C01818=1241.105,-36.655,-38.316,-179.706,5.196,148.807
C01819=1241.110,-36.904,-38.303,-179.709,5.195,148.808
C01820=1241.115,-37.154,-38.290,-179.711,5.195,148.809
C01821=1241.121,-37.404,-38.277,-179.714,5.195,148.810
C01822=1241.125,-37.653,-38.263,-179.716,5.196,148.810
C01823=1241.131,-37.903,-38.250,-179.719,5.195,148.811
C01824=1241.135,-38.153,-38.237,-179.721,5.195,148.812
C01825=1241.140,-38.402,-38.224,-179.724,5.195,148.813
C01826=1241.146,-38.651,-38.211,-179.726,5.194,148.813
C01827=1241.150,-38.901,-38.198,-179.728,5.195,148.814
C01828=1241.156,-39.151,-38.184,-179.731,5.194,148.815
C01829=1241.161,-39.401,-38.171,-179.733,5.194,148.815
C01830=1241.166,-39.649,-38.158,-179.736,5.194,148.816
C01831=1241.171,-39.900,-38.144,-179.738,5.195,148.817
C01832=1241.176,-40.149,-38.132,-179.741,5.194,148.818
C01833=1241.181,-40.398,-38.119,-179.743,5.194,148.818
C01834=1241.186,-40.649,-38.106,-179.746,5.194,148.819
C01835=1241.191,-40.898,-38.093,-179.749,5.193,148.820
C01836=1241.196,-41.148,-38.079,-179.751,5.194,148.820
C01837=1241.202,-41.397,-38.066,-179.753,5.193,148.821
C01838=1241.207,-41.646,-38.054,-179.755,5.194,148.822
C01839=1241.212,-41.897,-38.040,-179.758,5.193,148.823
C01840=1241.217,-42.146,-38.027,-179.760,5.193,148.823
C01841=1241.222,-42.396,-38.015,-179.763,5.193,148.824
C01842=1241.227,-42.645,-38.002,-179.765,5.194,148.825
C01843=1241.232,-42.894,-37.988,-179.768,5.193,148.826
C01844=1241.237,-43.144,-37.975,-179.771,5.193,148.826
C01845=1241.242,-43.394,-37.962,-179.773,5.193,148.827
C01846=1241.248,-43.643,-37.949,-179.775,5.192,148.828
C01847=1241.252,-43.893,-37.936,-179.778,5.193,148.828
C01848=1241.257,-44.143,-37.924,-179.780,5.192,148.829
C01849=1241.263,-44.393,-37.910,-179.782,5.192,148.830
C01850=1241.268,-44.642,-37.898,-179.785,5.192,148.831
C01851=1241.273,-44.892,-37.885,-179.788,5.193,148.831
C01852=1241.277,-45.142,-37.872,-179.790,5.192,148.832
C01853=1241.283,-45.391,-37.859,-179.793,5.192,148.833
C01854=1241.288,-45.641,-37.846,-179.795,5.192,148.834
C01855=1241.293,-45.891,-37.833,-179.798,5.191,148.834
C01856=1241.298,-46.140,-37.821,-179.800,5.192,148.835
C01857=1241.304,-46.389,-37.807,-179.802,5.191,148.836
C01858=1241.308,-46.640,-37.794,-179.804,5.192,148.836
C01859=1241.314,-46.889,-37.782,-179.807,5.191,148.837
C01860=1241.319,-47.138,-37.769,-179.809,5.191,148.838
C01861=1241.323,-47.388,-37.756,-179.812,5.191,148.839
C01862=1241.329,-47.638,-37.743,-179.814,5.192,148.839
C01863=1241.334,-47.908,-37.729,-179.817,5.191,148.840
C01864=1241.340,-48.177,-37.715,-179.820,5.191,148.841
C01865=1241.345,-48.447,-37.702,-179.822,5.191,148.842
C01866=1241.350,-48.716,-37.688,-179.825,5.191,148.842
C01867=1241.356,-48.966,-37.675,-179.828,5.190,148.843
C01868=1241.361,-49.215,-37.662,-179.830,5.191,148.844
C01869=1241.367,-49.465,-37.650,-179.832,5.190,148.845
C01870=1241.371,-49.715,-37.637,-179.835,5.190,148.845
C01871=1241.376,-49.964,-37.624,-179.838,5.190,148.846
C01872=1241.381,-50.213,-37.612,-179.840,5.191,148.847
C01873=1241.387,-50.464,-37.598,-179.842,5.190,148.848
C01874=1241.392,-50.713,-37.585,-179.845,5.190,148.848
C01875=1241.397,-50.963,-37.573,-179.847,5.190,148.849
C01876=1241.402,-51.212,-37.561,-179.849,5.190,148.850
C01877=1241.407,-51.462,-37.548,-179.852,5.190,148.850
C01878=1241.412,-51.711,-37.535,-179.854,5.190,148.851
C01879=1241.417,-51.961,-37.523,-179.857,5.190,148.852
C01880=1241.422,-52.210,-37.510,-179.859,5.189,148.853
C01881=1241.427,-52.460,-37.497,-179.862,5.190,148.853
C01882=1241.433,-52.710,-37.485,-179.865,5.189,148.854
C01883=1241.438,-52.960,-37.472,-179.867,5.190,148.855
C01884=1241.443,-53.209,-37.459,-179.869,5.189,148.856
C01885=1241.448,-53.459,-37.447,-179.871,5.189,148.856
C01886=1241.453,-53.708,-37.434,-179.874,5.189,148.857
C01887=1241.458,-53.958,-37.422,-179.876,5.189,148.858
C01888=1241.463,-54.208,-37.409,-179.879,5.189,148.858
C01889=1241.468,-54.458,-37.396,-179.881,5.189,148.859
C01890=1241.473,-54.707,-37.384,-179.884,5.189,148.860
C01891=1241.478,-54.956,-37.371,-179.886,5.189,148.861
C01892=1241.484,-55.206,-37.359,-179.889,5.189,148.861
C01893=1241.489,-55.456,-37.346,-179.891,5.189,148.862
C01894=1241.494,-55.706,-37.333,-179.894,5.189,148.863
C01895=1241.499,-55.955,-37.321,-179.896,5.189,148.864
C01896=1241.504,-56.205,-37.309,-179.898,5.188,148.864
C01897=1241.510,-56.454,-37.296,-179.901,5.189,148.865
C01898=1241.515,-56.704,-37.284,-179.903,5.188,148.866
C01899=1241.520,-56.954,-37.271,-179.906,5.188,148.866
C01900=1241.525,-57.204,-37.259,-179.908,5.188,148.867
C01901=1241.530,-57.453,-37.246,-179.911,5.188,148.868
C01902=1241.535,-57.703,-37.234,-179.913,5.188,148.869
C01903=1241.540,-57.952,-37.222,-179.916,5.188,148.869
C01904=1241.545,-58.202,-37.209,-179.918,5.188,148.870
C01905=1241.550,-58.452,-37.197,-179.921,5.188,148.871
C01906=1241.555,-58.702,-37.184,-179.923,5.188,148.872
C01907=1241.561,-58.951,-37.172,-179.925,5.187,148.872
C01908=1241.566,-59.201,-37.160,-179.927,5.188,148.873
C01909=1241.571,-59.450,-37.147,-179.930,5.187,148.874
C01910=1241.576,-59.699,-37.134,-179.932,5.188,148.874
C01911=1241.581,-59.950,-37.122,-179.935,5.187,148.875
C01912=1241.586,-60.199,-37.110,-179.937,5.188,148.876
C01913=1241.591,-60.448,-37.098,-179.940,5.187,148.877
C01914=1241.596,-60.698,-37.086,-179.942,5.188,148.877
C01915=1241.601,-60.948,-37.073,-179.945,5.187,148.878
C01916=1241.607,-61.198,-37.061,-179.947,5.187,148.879
C01917=1241.612,-61.447,-37.049,-179.950,5.187,148.880
C01918=1241.617,-61.697,-37.037,-179.952,5.187,148.880
C01919=1241.622,-61.947,-37.024,-179.954,5.187,148.881
C01920=1241.627,-62.196,-37.011,-179.957,5.187,148.882
C01921=1241.632,-62.446,-36.999,-179.959,5.187,148.882
C01922=1241.637,-62.695,-36.987,-179.961,5.187,148.883
C01923=1241.643,-62.945,-36.975,-179.964,5.187,148.884
C01924=1241.648,-63.195,-36.962,-179.967,5.187,148.885
C01925=1241.653,-63.444,-36.951,-179.969,5.187,148.885
C01926=1241.658,-63.694,-36.938,-179.971,5.187,148.886
C01927=1241.663,-63.944,-36.926,-179.974,5.187,148.887
C01928=1241.668,-64.193,-36.914,-179.976,5.187,148.888
C01929=1241.673,-64.444,-36.902,-179.979,5.186,148.888
C01930=1241.678,-64.693,-36.889,-179.981,5.187,148.889
C01931=1241.684,-64.943,-36.877,-179.983,5.186,148.890
C01932=1241.689,-65.192,-36.864,-179.986,5.187,148.890
C01933=1241.693,-65.442,-36.853,-179.988,5.186,148.891
C01934=1241.699,-65.691,-36.841,-179.991,5.187,148.892
C01935=1241.704,-65.941,-36.829,-179.993,5.186,148.893
C01936=1241.709,-66.190,-36.816,-179.996,5.187,148.893
C01937=1241.714,-66.440,-36.804,-179.998,5.186,148.894
C01938=1241.720,-66.690,-36.792,179.999,5.186,148.895
C01939=1241.724,-66.939,-36.780,179.997,5.186,148.896
C01940=1241.730,-67.189,-36.768,179.994,5.185,148.896
C01941=1241.735,-67.438,-36.756,179.992,5.186,148.897
C01942=1241.740,-67.688,-36.744,179.990,5.185,148.898
C01943=1241.746,-67.938,-36.732,179.987,5.186,148.898
C01944=1241.750,-68.187,-36.720,179.985,5.185,148.899
C01945=1241.756,-68.437,-36.708,179.982,5.186,148.900
C01946=1241.760,-68.687,-36.695,179.980,5.185,148.901
C01947=1241.765,-68.937,-36.683,179.977,5.186,148.901
C01948=1241.770,-69.187,-36.672,179.975,5.185,148.902
C01949=1241.775,-69.436,-36.659,179.973,5.186,148.903
C01950=1241.781,-69.686,-36.648,179.970,5.185,148.904
C01951=1241.786,-69.936,-36.636,179.968,5.185,148.904
C01952=1241.791,-70.185,-36.624,179.965,5.185,148.905
C01953=1241.796,-70.435,-36.612,179.963,5.185,148.906
C01954=1241.801,-70.685,-36.600,179.961,5.185,148.906
C01955=1241.807,-70.934,-36.587,179.958,5.185,148.907
C01956=1241.811,-71.184,-36.576,179.956,5.185,148.908
C01957=1241.817,-71.434,-36.564,179.953,5.185,148.909
C01958=1241.822,-71.683,-36.552,179.951,5.186,148.909
C01959=1241.827,-71.933,-36.540,179.948,5.185,148.910
C01960=1241.832,-72.183,-36.528,179.946,5.186,148.911
C01961=1241.837,-72.433,-36.516,179.944,5.185,148.912
C01962=1241.842,-72.682,-36.504,179.942,5.185,148.912
C01963=1241.847,-72.932,-36.493,179.939,5.185,148.913
C01964=1241.853,-73.181,-36.481,179.937,5.185,148.914
C01965=1241.859,-73.431,-36.469,179.934,5.185,148.914
C01966=1241.863,-73.680,-36.457,179.932,5.185,148.915
C01967=1241.868,-73.950,-36.444,179.929,5.185,148.916
C01968=1241.874,-74.221,-36.432,179.926,5.184,148.917
C01969=1241.881,-74.491,-36.419,179.924,5.185,148.917
C01970=1241.886,-74.761,-36.406,179.921,5.185,148.918
C01971=1241.891,-75.011,-36.394,179.919,5.185,148.919
C01972=1241.896,-75.260,-36.382,179.916,5.185,148.920
C01973=1241.900,-75.510,-36.371,179.914,5.185,148.921
C01974=1241.906,-75.760,-36.359,179.911,5.184,148.921
C01975=1241.911,-76.010,-36.347,179.909,5.185,148.922
C01976=1241.916,-76.259,-36.336,179.907,5.184,148.923
C01977=1241.921,-76.509,-36.324,179.905,5.185,148.923
C01978=1241.927,-76.758,-36.311,179.902,5.184,148.924
C01979=1241.932,-77.008,-36.300,179.900,5.184,148.925
C01980=1241.937,-77.258,-36.288,179.897,5.184,148.925
C01981=1241.942,-77.507,-36.277,179.895,5.184,148.926
C01982=1241.947,-77.757,-36.265,179.892,5.184,148.927
C01983=1241.953,-78.007,-36.253,179.890,5.185,148.928
C01984=1241.957,-78.257,-36.242,179.887,5.184,148.929
C01985=1241.963,-78.507,-36.230,179.885,5.184,148.929
C01986=1241.967,-78.756,-36.218,179.882,5.184,148.930
C01987=1241.973,-79.006,-36.206,179.880,5.184,148.931
C01988=1241.979,-79.255,-36.195,179.878,5.184,148.931
C01989=1241.983,-79.504,-36.183,179.875,5.184,148.932
C01990=1241.989,-79.754,-36.171,179.873,5.184,148.933
C01991=1241.994,-80.004,-36.160,179.871,5.184,148.934
C01992=1241.999,-80.254,-36.148,179.868,5.184,148.934
C01993=1242.004,-80.504,-36.137,179.866,5.184,148.935
C01994=1242.009,-80.753,-36.125,179.863,5.183,148.936
C01995=1242.014,-81.003,-36.114,179.861,5.184,148.936
C01996=1242.020,-81.252,-36.102,179.859,5.184,148.937
C01997=1242.025,-81.502,-36.091,179.856,5.184,148.938
C01998=1242.030,-81.752,-36.079,179.854,5.184,148.939
C01999=1242.035,-82.001,-36.068,179.851,5.184,148.939
C02000=1242.040,-82.251,-36.056,179.849,5.184,148.940
C02001=1242.045,-82.501,-36.045,179.846,5.184,148.941
C02002=1242.050,-82.751,-36.033,179.844,5.184,148.942
C02003=1242.055,-83.000,-36.022,179.842,5.184,148.942
C02004=1242.061,-83.250,-36.010,179.840,5.184,148.943
C02005=1242.066,-83.499,-35.999,179.837,5.183,148.944
C02006=1242.071,-83.749,-35.987,179.835,5.184,148.944
C02007=1242.076,-83.999,-35.975,179.832,5.183,148.945
C02008=1242.081,-84.249,-35.964,179.830,5.184,148.946
C02009=1242.086,-84.498,-35.953,179.827,5.183,148.947
C02010=1242.092,-84.748,-35.941,179.825,5.184,148.947
C02011=1242.097,-84.997,-35.929,179.823,5.183,148.948
C02012=1242.102,-85.247,-35.918,179.820,5.183,148.949
C02013=1242.107,-85.498,-35.907,179.818,5.183,148.949
C02014=1242.113,-85.747,-35.895,179.815,5.184,148.950
C02015=1242.118,-85.997,-35.884,179.813,5.183,148.951
C02016=1242.122,-86.246,-35.873,179.810,5.184,148.952
C02017=1242.128,-86.496,-35.861,179.808,5.184,148.952
C02018=1242.133,-86.746,-35.850,179.806,5.183,148.953
C02019=1242.139,-86.995,-35.838,179.804,5.184,148.954
C02020=1242.143,-87.245,-35.827,179.801,5.183,148.955
C02021=1242.148,-87.495,-35.816,179.799,5.184,148.955
C02022=1242.154,-87.745,-35.804,179.796,5.183,148.956
C02023=1242.159,-87.994,-35.794,179.794,5.184,148.957
C02024=1242.164,-88.244,-35.782,179.791,5.183,148.957
C02025=1242.169,-88.493,-35.770,179.789,5.183,148.958
C02026=1242.174,-88.743,-35.759,179.787,5.183,148.959
C02027=1242.180,-88.993,-35.748,179.785,5.183,148.960
C02028=1242.185,-89.242,-35.737,179.782,5.183,148.960
C02029=1242.190,-89.492,-35.725,179.780,5.183,148.961
C02030=1242.195,-89.742,-35.714,179.777,5.183,148.962
C02031=1242.200,-89.992,-35.703,179.775,5.183,148.962
C02032=1242.206,-90.241,-35.692,179.772,5.183,148.963
C02033=1242.211,-90.491,-35.680,179.770,5.183,148.964
C02034=1242.215,-90.741,-35.669,179.768,5.184,148.965
C02035=1242.221,-90.990,-35.658,179.765,5.183,148.965
C02036=1242.226,-91.240,-35.647,179.763,5.184,148.966
C02037=1242.231,-91.490,-35.636,179.760,5.183,148.967
C02038=1242.236,-91.740,-35.624,179.758,5.183,148.968
C02039=1242.242,-91.989,-35.613,179.755,5.183,148.968
C02040=1242.247,-92.239,-35.602,179.753,5.183,148.969
C02041=1242.251,-92.488,-35.591,179.751,5.183,148.970
C02042=1242.257,-92.738,-35.579,179.749,5.183,148.970
C02043=1242.262,-92.988,-35.569,179.746,5.183,148.971
C02044=1242.267,-93.238,-35.558,179.744,5.183,148.972
C02045=1242.273,-93.488,-35.546,179.741,5.183,148.973
C02046=1242.278,-93.737,-35.536,179.739,5.183,148.973
C02047=1242.283,-93.987,-35.524,179.737,5.183,148.974
C02048=1242.288,-94.236,-35.513,179.734,5.183,148.975
C02049=1242.294,-94.486,-35.502,179.732,5.183,148.975
C02050=1242.299,-94.736,-35.491,179.729,5.183,148.976
C02051=1242.303,-94.985,-35.480,179.727,5.183,148.977
C02052=1242.310,-95.235,-35.469,179.725,5.183,148.978
C02053=1242.314,-95.485,-35.458,179.723,5.183,148.978
C02054=1242.319,-95.735,-35.446,179.720,5.183,148.979
C02055=1242.325,-95.984,-35.436,179.718,5.183,148.980
C02056=1242.329,-96.234,-35.425,179.715,5.183,148.981
C02057=1242.335,-96.484,-35.414,179.713,5.183,148.981
C02058=1242.340,-96.733,-35.403,179.710,5.183,148.982
C02059=1242.345,-96.983,-35.391,179.708,5.183,148.983
C02060=1242.350,-97.233,-35.381,179.706,5.183,148.984
C02061=1242.356,-97.482,-35.369,179.703,5.183,148.984
C02062=1242.361,-97.733,-35.359,179.701,5.183,148.985
C02063=1242.366,-97.982,-35.347,179.698,5.183,148.986
C02064=1242.371,-98.232,-35.337,179.696,5.183,148.986
C02065=1242.376,-98.481,-35.326,179.693,5.183,148.987
C02066=1242.381,-98.731,-35.314,179.691,5.183,148.988
C02067=1242.387,-98.981,-35.304,179.689,5.183,148.989
C02068=1242.392,-99.230,-35.293,179.687,5.183,148.989
C02069=1242.397,-99.480,-35.282,179.684,5.182,148.990
C02070=1242.402,-99.730,-35.271,179.682,5.183,148.991
C02071=1242.408,-100.001,-35.259,179.679,5.182,148.991
C02072=1242.414,-100.271,-35.248,179.677,5.183,148.992
C02073=1242.419,-100.542,-35.236,179.674,5.183,148.993
C02074=1242.425,-100.813,-35.224,179.672,5.183,148.994
C02075=1242.430,-101.063,-35.213,179.669,5.183,148.994
C02076=1242.435,-101.312,-35.202,179.667,5.183,148.995
C02077=1242.440,-101.563,-35.192,179.664,5.182,148.996
C02078=1242.445,-101.811,-35.181,179.662,5.183,148.997
C02079=1242.450,-102.062,-35.170,179.660,5.182,148.997
C02080=1242.456,-102.311,-35.159,179.657,5.183,148.998
C02081=1242.461,-102.561,-35.148,179.655,5.182,148.999
C02082=1242.467,-102.810,-35.137,179.653,5.183,148.999
C02083=1242.472,-103.060,-35.127,179.651,5.183,149.000
C02084=1242.477,-103.311,-35.116,179.648,5.183,149.001
C02085=1242.482,-103.560,-35.105,179.646,5.183,149.002
C02086=1242.487,-103.810,-35.094,179.643,5.182,149.002
C02087=1242.492,-104.059,-35.084,179.641,5.183,149.003
C02088=1242.497,-104.309,-35.073,179.638,5.182,149.004
C02089=1242.503,-104.558,-35.063,179.636,5.183,149.004
C02090=1242.507,-104.808,-35.051,179.634,5.182,149.005
C02091=1242.513,-105.058,-35.041,179.632,5.183,149.006
C02092=1242.518,-105.308,-35.031,179.629,5.182,149.007
C02093=1242.523,-105.558,-35.019,179.627,5.182,149.007
C02094=1242.529,-105.807,-35.009,179.625,5.183,149.008
C02095=1242.534,-106.057,-34.997,179.622,5.182,149.009
C02096=1242.539,-106.307,-34.987,179.620,5.183,149.009
C02097=1242.544,-106.557,-34.977,179.617,5.182,149.010
C02098=1242.550,-106.806,-34.966,179.615,5.183,149.011
C02099=1242.555,-107.056,-34.955,179.612,5.182,149.012
C02100=1242.560,-107.305,-34.945,179.610,5.183,149.012
C02101=1242.565,-107.556,-34.934,179.608,5.182,149.013
C02102=1242.571,-107.805,-34.923,179.606,5.182,149.014
C02103=1242.576,-108.055,-34.913,179.603,5.183,149.014
C02104=1242.581,-108.304,-34.903,179.601,5.182,149.015
C02105=1242.586,-108.554,-34.891,179.599,5.183,149.016
C02106=1242.591,-108.804,-34.881,179.596,5.183,149.017
C02107=1242.596,-109.054,-34.870,179.593,5.183,149.018
C02108=1242.602,-109.303,-34.860,179.591,5.183,149.018
C02109=1242.607,-109.553,-34.849,179.589,5.183,149.019
C02110=1242.612,-109.803,-34.839,179.586,5.182,149.020
C02111=1242.617,-110.053,-34.828,179.584,5.183,149.020
C02112=1242.622,-110.302,-34.819,179.582,5.183,149.021
C02113=1242.627,-110.552,-34.807,179.580,5.182,149.022
C02114=1242.632,-110.801,-34.797,179.578,5.183,149.022
C02115=1242.637,-111.051,-34.786,179.575,5.182,149.023
C02116=1242.643,-111.301,-34.776,179.573,5.183,149.024
C02117=1242.648,-111.551,-34.766,179.570,5.182,149.024
C02118=1242.654,-111.801,-34.755,179.568,5.183,149.025
C02119=1242.659,-112.050,-34.745,179.565,5.182,149.026
C02120=1242.664,-112.300,-34.734,179.563,5.182,149.027
C02121=1242.670,-112.549,-34.724,179.561,5.183,149.027
C02122=1242.675,-112.800,-34.713,179.558,5.182,149.028
C02123=1242.680,-113.049,-34.703,179.556,5.183,149.029
C02124=1242.685,-113.300,-34.692,179.554,5.182,149.029
C02125=1242.690,-113.548,-34.682,179.552,5.183,149.030
C02126=1242.695,-113.798,-34.672,179.549,5.182,149.031
C02127=1242.700,-114.048,-34.661,179.547,5.183,149.032
C02128=1242.706,-114.297,-34.651,179.544,5.182,149.032
C02129=1242.711,-114.548,-34.641,179.542,5.182,149.033
C02130=1242.716,-114.797,-34.630,179.540,5.183,149.034
C02131=1242.721,-115.048,-34.620,179.537,5.182,149.035
C02132=1242.727,-115.297,-34.610,179.535,5.183,149.035
C02133=1242.732,-115.546,-34.600,179.532,5.182,149.036
C02134=1242.737,-115.796,-34.589,179.530,5.183,149.037
C02135=1242.742,-116.045,-34.578,179.528,5.182,149.037
C02136=1242.747,-116.296,-34.568,179.526,5.183,149.038
C02137=1242.753,-116.545,-34.558,179.523,5.182,149.039
C02138=1242.758,-116.795,-34.547,179.521,5.183,149.040
C02139=1242.763,-117.045,-34.537,179.519,5.183,149.040
C02140=1242.768,-117.294,-34.527,179.516,5.182,149.041
C02141=1242.773,-117.545,-34.517,179.514,5.183,149.042
C02142=1242.779,-117.794,-34.506,179.511,5.182,149.042
C02143=1242.784,-118.044,-34.496,179.509,5.183,149.043
C02144=1242.789,-118.294,-34.486,179.506,5.182,149.044
C02145=1242.794,-118.543,-34.476,179.504,5.183,149.045
C02146=1242.799,-118.793,-34.465,179.502,5.182,149.045
C02147=1242.805,-119.043,-34.455,179.500,5.183,149.046
C02148=1242.811,-119.292,-34.445,179.497,5.183,149.047
C02149=1242.815,-119.542,-34.435,179.495,5.182,149.047
C02150=1242.820,-119.792,-34.425,179.493,5.183,149.048
C02151=1242.826,-120.041,-34.415,179.490,5.182,149.049
C02152=1242.831,-120.292,-34.404,179.488,5.183,149.050
C02153=1242.836,-120.541,-34.394,179.485,5.182,149.050
C02154=1242.841,-120.790,-34.384,179.483,5.183,149.051
C02155=1242.846,-121.041,-34.374,179.481,5.183,149.052
C02156=1242.852,-121.290,-34.363,179.478,5.183,149.052
C02157=1242.857,-121.539,-34.354,179.476,5.183,149.053
C02158=1242.862,-121.790,-34.344,179.474,5.183,149.054
C02159=1242.868,-122.040,-34.334,179.472,5.183,149.055
C02160=1242.873,-122.289,-34.324,179.469,5.182,149.055
C02161=1242.878,-122.539,-34.314,179.467,5.182,149.056
C02162=1242.883,-122.789,-34.303,179.465,5.182,149.056
C02163=1242.889,-123.038,-34.293,179.462,5.182,149.057
C02164=1242.893,-123.288,-34.283,179.460,5.183,149.058
C02165=1242.899,-123.538,-34.273,179.458,5.182,149.059
C02166=1242.904,-123.787,-34.263,179.456,5.183,149.059
C02167=1242.909,-124.037,-34.254,179.453,5.182,149.060
C02168=1242.914,-124.288,-34.243,179.451,5.183,149.061
C02169=1242.920,-124.537,-34.233,179.448,5.182,149.062
C02170=1242.925,-124.786,-34.224,179.446,5.183,149.062
C02171=1242.930,-125.037,-34.213,179.444,5.183,149.063
C02172=1242.936,-125.286,-34.203,179.441,5.183,149.064
C02173=1242.941,-125.536,-34.194,179.439,5.183,149.064
C02174=1242.946,-125.786,-34.184,179.436,5.182,149.065
C02175=1242.524,-125.796,-34.218,179.432,5.186,149.067
C02176=1242.519,-125.547,-34.227,179.435,5.186,149.067
C02177=1242.514,-125.297,-34.237,179.437,5.186,149.066
C02178=1242.509,-125.047,-34.248,179.439,5.186,149.065
C02179=1242.504,-124.798,-34.258,179.442,5.186,149.064
C02180=1242.498,-124.548,-34.268,179.444,5.186,149.064
C02181=1242.493,-124.297,-34.278,179.446,5.186,149.063
C02182=1242.488,-124.048,-34.287,179.448,5.186,149.062
C02183=1242.482,-123.799,-34.297,179.451,5.186,149.061
C02184=1242.477,-123.548,-34.308,179.453,5.186,149.061
C02185=1242.472,-123.299,-34.318,179.455,5.185,149.060
C02186=1242.467,-123.050,-34.328,179.458,5.186,149.059
C02187=1242.461,-122.800,-34.338,179.460,5.186,149.059
C02188=1242.456,-122.549,-34.348,179.463,5.186,149.058
C02189=1242.451,-122.300,-34.358,179.465,5.186,149.057
C02190=1242.446,-122.050,-34.368,179.468,5.186,149.056
C02191=1242.441,-121.800,-34.378,179.470,5.186,149.056
C02192=1242.435,-121.551,-34.389,179.472,5.186,149.055
C02193=1242.430,-121.301,-34.398,179.474,5.186,149.054
C02194=1242.425,-121.051,-34.409,179.476,5.186,149.054
C02195=1242.420,-120.802,-34.419,179.479,5.186,149.053
C02196=1242.415,-120.552,-34.429,179.481,5.186,149.052
C02197=1242.410,-120.302,-34.439,179.483,5.186,149.052
C02198=1242.404,-120.053,-34.449,179.486,5.186,149.051
C02199=1242.398,-119.803,-34.460,179.488,5.186,149.050
C02200=1242.393,-119.553,-34.470,179.490,5.186,149.050
C02201=1242.388,-119.303,-34.479,179.492,5.186,149.049
C02202=1242.383,-119.053,-34.489,179.495,5.186,149.048
C02203=1242.378,-118.803,-34.500,179.497,5.186,149.047
C02204=1242.372,-118.554,-34.510,179.500,5.186,149.047
C02205=1242.368,-118.304,-34.520,179.502,5.186,149.046
C02206=1242.362,-118.054,-34.530,179.505,5.186,149.045
C02207=1242.357,-117.805,-34.540,179.507,5.186,149.045
C02208=1242.352,-117.554,-34.551,179.509,5.186,149.044
C02209=1242.346,-117.305,-34.562,179.512,5.186,149.043
C02210=1242.342,-117.056,-34.572,179.514,5.186,149.042
C02211=1242.337,-116.806,-34.582,179.516,5.186,149.042
C02212=1242.331,-116.556,-34.592,179.518,5.186,149.041
C02213=1242.326,-116.306,-34.603,179.521,5.186,149.040
C02214=1242.320,-116.057,-34.613,179.523,5.186,149.039
C02215=1242.315,-115.807,-34.623,179.526,5.186,149.039
C02216=1242.310,-115.557,-34.633,179.528,5.186,149.038
C02217=1242.305,-115.308,-34.644,179.531,5.186,149.037
C02218=1242.300,-115.057,-34.654,179.533,5.186,149.037
C02219=1242.294,-114.808,-34.664,179.535,5.186,149.036
C02220=1242.289,-114.558,-34.674,179.538,5.186,149.035
C02221=1242.284,-114.308,-34.685,179.540,5.186,149.034
C02222=1242.278,-114.058,-34.695,179.542,5.186,149.034
C02223=1242.274,-113.809,-34.706,179.544,5.186,149.033
C02224=1242.269,-113.560,-34.716,179.547,5.186,149.032
C02225=1242.264,-113.309,-34.727,179.549,5.186,149.032
C02226=1242.258,-113.060,-34.737,179.552,5.186,149.031
C02227=1242.252,-112.810,-34.747,179.554,5.186,149.030
C02228=1242.247,-112.560,-34.758,179.556,5.185,149.029
C02229=1242.242,-112.310,-34.768,179.559,5.186,149.029
C02230=1242.237,-112.061,-34.779,179.561,5.186,149.028
C02231=1242.231,-111.811,-34.789,179.563,5.186,149.027
C02232=1242.226,-111.561,-34.800,179.566,5.186,149.027
C02233=1242.222,-111.312,-34.810,179.568,5.186,149.026
C02234=1242.217,-111.062,-34.820,179.570,5.186,149.025
C02235=1242.211,-110.812,-34.830,179.573,5.186,149.024
C02236=1242.206,-110.563,-34.841,179.575,5.186,149.024
C02237=1242.201,-110.313,-34.852,179.577,5.185,149.023
C02238=1242.195,-110.063,-34.862,179.580,5.186,149.022
C02239=1242.190,-109.813,-34.873,179.582,5.186,149.022
C02240=1242.185,-109.564,-34.884,179.585,5.186,149.021
C02241=1242.180,-109.314,-34.894,179.586,5.186,149.020
C02242=1242.174,-109.064,-34.904,179.589,5.186,149.020
C02243=1242.169,-108.814,-34.915,179.591,5.186,149.019
C02244=1242.164,-108.565,-34.926,179.594,5.187,149.018
C02245=1242.159,-108.315,-34.936,179.596,5.186,149.018
C02246=1242.153,-108.065,-34.947,179.598,5.186,149.017
C02247=1242.148,-107.815,-34.957,179.601,5.186,149.016
C02248=1242.143,-107.566,-34.968,179.603,5.186,149.015
C02249=1242.138,-107.316,-34.979,179.606,5.186,149.014
C02250=1242.132,-107.066,-34.989,179.608,5.186,149.014
C02251=1242.128,-106.817,-35.000,179.611,5.186,149.013
C02252=1242.122,-106.567,-35.010,179.613,5.186,149.012
C02253=1242.117,-106.317,-35.021,179.615,5.186,149.012
C02254=1242.112,-106.068,-35.032,179.617,5.186,149.011
C02255=1242.107,-105.818,-35.043,179.620,5.186,149.010
C02256=1242.102,-105.568,-35.053,179.622,5.186,149.009
C02257=1242.097,-105.319,-35.064,179.624,5.186,149.009
C02258=1242.092,-105.068,-35.075,179.627,5.186,149.008
C02259=1242.086,-104.819,-35.085,179.629,5.186,149.007
C02260=1242.081,-104.569,-35.096,179.632,5.186,149.007
C02261=1242.076,-104.320,-35.106,179.634,5.186,149.006
C02262=1242.071,-104.070,-35.117,179.637,5.186,149.005
C02263=1242.065,-103.821,-35.128,179.639,5.186,149.004
C02264=1242.060,-103.570,-35.139,179.641,5.186,149.004
C02265=1242.054,-103.321,-35.150,179.643,5.186,149.003
C02266=1242.049,-103.071,-35.161,179.646,5.186,149.002
C02267=1242.044,-102.821,-35.171,179.648,5.186,149.002
C02268=1242.039,-102.572,-35.182,179.650,5.186,149.001
C02269=1242.034,-102.321,-35.193,179.653,5.186,149.000
C02270=1242.029,-102.073,-35.203,179.655,5.186,148.999
C02271=1242.024,-101.822,-35.214,179.658,5.186,148.999
C02272=1242.019,-101.573,-35.225,179.660,5.186,148.998
C02273=1242.013,-101.323,-35.236,179.663,5.186,148.997
C02274=1242.008,-101.073,-35.247,179.665,5.186,148.997
C02275=1242.002,-100.824,-35.258,179.667,5.186,148.996
C02276=1241.998,-100.553,-35.269,179.669,5.186,148.995
C02277=1241.992,-100.282,-35.282,179.672,5.187,148.994
C02278=1241.985,-100.011,-35.293,179.675,5.186,148.994
C02279=1241.981,-99.740,-35.304,179.677,5.186,148.993
C02280=1241.976,-99.491,-35.316,179.679,5.186,148.992
C02281=1241.970,-99.241,-35.326,179.682,5.186,148.991
C02282=1241.965,-98.991,-35.338,179.684,5.186,148.991
C02283=1241.960,-98.741,-35.348,179.687,5.187,148.990
C02284=1241.955,-98.492,-35.359,179.689,5.186,148.989
C02285=1241.950,-98.242,-35.370,179.692,5.187,148.989
C02286=1241.944,-97.993,-35.381,179.694,5.186,148.988
C02287=1241.939,-97.742,-35.392,179.696,5.187,148.987
C02288=1241.934,-97.493,-35.403,179.699,5.186,148.986
C02289=1241.929,-97.244,-35.414,179.701,5.186,148.986
C02290=1241.924,-96.994,-35.425,179.703,5.186,148.985
C02291=1241.919,-96.744,-35.436,179.705,5.186,148.984
C02292=1241.913,-96.494,-35.447,179.708,5.187,148.984
C02293=1241.908,-96.245,-35.458,179.710,5.186,148.983
C02294=1241.903,-95.995,-35.469,179.713,5.187,148.982
C02295=1241.898,-95.745,-35.480,179.715,5.186,148.981
C02296=1241.892,-95.495,-35.492,179.718,5.187,148.981
C02297=1241.887,-95.245,-35.502,179.720,5.186,148.980
C02298=1241.882,-94.996,-35.513,179.723,5.187,148.979
C02299=1241.877,-94.747,-35.524,179.725,5.186,148.978
C02300=1241.871,-94.496,-35.535,179.728,5.187,148.978
C02301=1241.866,-94.247,-35.546,179.730,5.186,148.977
C02302=1241.861,-93.998,-35.558,179.732,5.186,148.976
C02303=1241.856,-93.747,-35.568,179.735,5.186,148.975
C02304=1241.850,-93.498,-35.580,179.737,5.186,148.975
C02305=1241.846,-93.248,-35.591,179.739,5.187,148.974
C02306=1241.841,-92.998,-35.602,179.741,5.186,148.973
C02307=1241.835,-92.749,-35.613,179.744,5.187,148.973
C02308=1241.830,-92.499,-35.624,179.746,5.186,148.972
C02309=1241.825,-92.249,-35.635,179.749,5.187,148.971
C02310=1241.820,-91.999,-35.646,179.751,5.186,148.970
C02311=1241.814,-91.750,-35.658,179.754,5.187,148.970
C02312=1241.810,-91.501,-35.669,179.756,5.187,148.969
C02313=1241.805,-91.250,-35.680,179.758,5.187,148.968
C02314=1241.799,-91.001,-35.691,179.760,5.187,148.968
C02315=1241.794,-90.751,-35.703,179.763,5.187,148.967
C02316=1241.789,-90.501,-35.713,179.765,5.187,148.966
C02317=1241.783,-90.251,-35.725,179.767,5.186,148.965
C02318=1241.778,-90.002,-35.736,179.770,5.187,148.965
C02319=1241.773,-89.753,-35.747,179.772,5.187,148.964
C02320=1241.768,-89.503,-35.759,179.775,5.187,148.963
C02321=1241.763,-89.253,-35.770,179.777,5.187,148.963
C02322=1241.757,-89.003,-35.781,179.780,5.187,148.962
C02323=1241.752,-88.754,-35.792,179.782,5.186,148.961
C02324=1241.748,-88.504,-35.804,179.785,5.187,148.960
C02325=1241.742,-88.254,-35.816,179.787,5.187,148.960
C02326=1241.737,-88.005,-35.826,179.790,5.187,148.959
C02327=1241.732,-87.755,-35.837,179.792,5.187,148.958
C02328=1241.726,-87.505,-35.849,179.794,5.187,148.957
C02329=1241.722,-87.255,-35.860,179.796,5.187,148.957
C02330=1241.716,-87.006,-35.872,179.799,5.187,148.956
C02331=1241.711,-86.757,-35.883,179.801,5.187,148.955
C02332=1241.706,-86.506,-35.894,179.804,5.187,148.955
C02333=1241.701,-86.256,-35.906,179.806,5.187,148.954
C02334=1241.696,-86.007,-35.917,179.808,5.187,148.953
C02335=1241.690,-85.757,-35.928,179.811,5.187,148.952
C02336=1241.685,-85.508,-35.940,179.813,5.187,148.952
C02337=1241.680,-85.258,-35.952,179.815,5.187,148.951
C02338=1241.675,-85.008,-35.963,179.818,5.187,148.950
C02339=1241.670,-84.759,-35.974,179.820,5.187,148.950
C02340=1241.664,-84.509,-35.986,179.822,5.187,148.949
C02341=1241.660,-84.260,-35.997,179.825,5.187,148.948
C02342=1241.654,-84.009,-36.008,179.828,5.187,148.947
C02343=1241.649,-83.760,-36.019,179.830,5.187,148.947
C02344=1241.644,-83.510,-36.031,179.832,5.187,148.946
C02345=1241.639,-83.260,-36.043,179.835,5.187,148.945
C02346=1241.633,-83.011,-36.054,179.837,5.187,148.944
C02347=1241.628,-82.761,-36.065,179.840,5.188,148.944
C02348=1241.623,-82.511,-36.077,179.842,5.187,148.943
C02349=1241.618,-82.262,-36.089,179.845,5.188,148.942
C02350=1241.613,-82.012,-36.100,179.847,5.187,148.942
C02351=1241.608,-81.762,-36.112,179.849,5.188,148.941
C02352=1241.603,-81.512,-36.124,179.851,5.187,148.940
C02353=1241.597,-81.263,-36.135,179.854,5.188,148.939
C02354=1241.592,-81.013,-36.146,179.856,5.188,148.939
C02355=1241.587,-80.764,-36.158,179.858,5.187,148.938
C02356=1241.582,-80.514,-36.170,179.861,5.188,148.937
C02357=1241.577,-80.264,-36.181,179.864,5.187,148.936
C02358=1241.572,-80.014,-36.193,179.866,5.187,148.936
C02359=1241.567,-79.765,-36.204,179.868,5.187,148.935
C02360=1241.561,-79.515,-36.216,179.871,5.188,148.934
C02361=1241.557,-79.266,-36.228,179.873,5.187,148.934
C02362=1241.551,-79.016,-36.239,179.876,5.188,148.933
C02363=1241.546,-78.766,-36.251,179.878,5.187,148.932
C02364=1241.541,-78.517,-36.263,179.880,5.188,148.931
C02365=1241.536,-78.267,-36.275,179.883,5.188,148.931
C02366=1241.531,-78.017,-36.286,179.885,5.188,148.930
C02367=1241.526,-77.767,-36.298,179.887,5.188,148.929
C02368=1241.520,-77.517,-36.310,179.890,5.188,148.929
C02369=1241.515,-77.268,-36.321,179.892,5.188,148.928
C02370=1241.509,-77.018,-36.332,179.895,5.188,148.927
C02371=1241.505,-76.769,-36.344,179.897,5.188,148.926
C02372=1241.500,-76.520,-36.356,179.900,5.188,148.925
C02373=1241.494,-76.270,-36.368,179.902,5.188,148.925
C02374=1241.489,-76.020,-36.379,179.905,5.188,148.924
C02375=1241.484,-75.770,-36.391,179.907,5.188,148.923
C02376=1241.479,-75.520,-36.403,179.910,5.188,148.923
C02377=1241.474,-75.270,-36.415,179.912,5.188,148.922
C02378=1241.469,-75.021,-36.427,179.914,5.188,148.921
C02379=1241.464,-74.772,-36.438,179.916,5.188,148.921
C02380=1241.458,-74.502,-36.451,179.919,5.189,148.920
C02381=1241.452,-74.231,-36.465,179.922,5.188,148.919
C02382=1241.447,-73.961,-36.478,179.924,5.188,148.918
C02383=1241.441,-73.691,-36.489,179.927,5.189,148.917
C02384=1241.436,-73.442,-36.501,179.929,5.189,148.917
C02385=1241.431,-73.192,-36.513,179.932,5.189,148.916
C02386=1241.425,-72.942,-36.525,179.934,5.188,148.915
C02387=1241.421,-72.692,-36.537,179.937,5.189,148.914
C02388=1241.416,-72.443,-36.549,179.939,5.188,148.914
C02389=1241.410,-72.193,-36.561,179.942,5.189,148.913
C02390=1241.405,-71.943,-36.572,179.944,5.189,148.912
C02391=1241.400,-71.693,-36.584,179.947,5.189,148.912
C02392=1241.395,-71.444,-36.597,179.949,5.189,148.911
C02393=1241.389,-71.194,-36.609,179.951,5.189,148.910
C02394=1241.385,-70.944,-36.620,179.953,5.189,148.909
C02395=1241.380,-70.695,-36.633,179.956,5.189,148.909
C02396=1241.374,-70.445,-36.644,179.958,5.189,148.908
C02397=1241.369,-70.195,-36.656,179.961,5.190,148.907
C02398=1241.364,-69.946,-36.668,179.963,5.189,148.906
C02399=1241.359,-69.696,-36.680,179.966,5.189,148.906
C02400=1241.354,-69.446,-36.692,179.968,5.189,148.905
C02401=1241.348,-69.197,-36.705,179.971,5.189,148.904
C02402=1241.344,-68.947,-36.716,179.973,5.189,148.904
C02403=1241.338,-68.697,-36.728,179.976,5.190,148.903
C02404=1241.333,-68.448,-36.740,179.978,5.189,148.902
C02405=1241.328,-68.198,-36.752,179.980,5.190,148.901
C02406=1241.323,-67.949,-36.764,179.982,5.189,148.901
C02407=1241.318,-67.699,-36.776,179.985,5.190,148.900
C02408=1241.312,-67.449,-36.788,179.987,5.190,148.899
C02409=1241.307,-67.200,-36.801,179.990,5.190,148.899
C02410=1241.302,-66.950,-36.813,179.993,5.189,148.898
C02411=1241.297,-66.700,-36.824,179.995,5.190,148.897
C02412=1241.292,-66.451,-36.837,179.997,5.190,148.896
C02413=1241.287,-66.201,-36.848,180.000,5.190,148.896
C02414=1241.282,-65.952,-36.861,-179.998,5.190,148.895
C02415=1241.277,-65.701,-36.873,-179.995,5.190,148.894
C02416=1241.272,-65.452,-36.886,-179.993,5.190,148.893
C02417=1241.267,-65.202,-36.897,-179.991,5.190,148.893
C02418=1241.262,-64.953,-36.910,-179.988,5.190,148.892
C02419=1241.256,-64.703,-36.922,-179.986,5.190,148.891
C02420=1241.251,-64.454,-36.934,-179.984,5.190,148.891
C02421=1241.246,-64.204,-36.946,-179.981,5.191,148.890
C02422=1241.240,-63.954,-36.958,-179.978,5.190,148.889
C02423=1241.235,-63.705,-36.971,-179.976,5.190,148.888
C02424=1241.231,-63.456,-36.983,-179.974,5.190,148.888
C02425=1241.225,-63.206,-36.994,-179.971,5.191,148.887
C02426=1241.220,-62.956,-37.007,-179.969,5.190,148.886
C02427=1241.215,-62.706,-37.019,-179.966,5.191,148.885
C02428=1241.210,-62.456,-37.032,-179.964,5.190,148.885
C02429=1241.205,-62.206,-37.044,-179.961,5.191,148.884
C02430=1241.200,-61.957,-37.056,-179.959,5.191,148.883
C02431=1241.194,-61.707,-37.068,-179.957,5.191,148.883
C02432=1241.189,-61.458,-37.081,-179.955,5.191,148.882
C02433=1241.184,-61.208,-37.093,-179.951,5.191,148.881
C02434=1241.179,-60.959,-37.105,-179.949,5.191,148.880
C02435=1241.174,-60.710,-37.117,-179.947,5.191,148.880
C02436=1241.169,-60.459,-37.130,-179.945,5.191,148.879
C02437=1241.164,-60.210,-37.142,-179.942,5.191,148.878
C02438=1241.159,-59.960,-37.154,-179.940,5.191,148.877
C02439=1241.154,-59.710,-37.167,-179.937,5.191,148.877
C02440=1241.149,-59.461,-37.179,-179.935,5.191,148.876
C02441=1241.143,-59.211,-37.191,-179.932,5.192,148.875
C02442=1241.138,-58.962,-37.204,-179.930,5.191,148.875
C02443=1241.134,-58.712,-37.217,-179.928,5.192,148.874
C02444=1241.128,-58.462,-37.229,-179.925,5.191,148.873
C02445=1241.123,-58.212,-37.241,-179.922,5.191,148.872
C02446=1241.118,-57.963,-37.253,-179.920,5.191,148.872
C02447=1241.112,-57.713,-37.266,-179.918,5.192,148.871
C02448=1241.107,-57.464,-37.278,-179.915,5.192,148.870
C02449=1241.103,-57.214,-37.291,-179.913,5.192,148.869
C02450=1241.097,-56.964,-37.303,-179.910,5.192,148.869
C02451=1241.092,-56.715,-37.316,-179.908,5.192,148.868
C02452=1241.087,-56.465,-37.328,-179.906,5.192,148.867
C02453=1241.082,-56.215,-37.340,-179.903,5.192,148.867
C02454=1241.077,-55.965,-37.353,-179.901,5.193,148.866
C02455=1241.072,-55.716,-37.366,-179.898,5.192,148.865
C02456=1241.067,-55.467,-37.378,-179.896,5.192,148.864
C02457=1241.062,-55.217,-37.390,-179.893,5.192,148.864
C02458=1241.056,-54.967,-37.403,-179.891,5.193,148.863
C02459=1241.052,-54.717,-37.416,-179.889,5.192,148.862
C02460=1241.047,-54.468,-37.429,-179.886,5.193,148.861
C02461=1241.041,-54.218,-37.440,-179.884,5.192,148.861
C02462=1241.036,-53.969,-37.453,-179.881,5.193,148.860
C02463=1241.031,-53.719,-37.467,-179.879,5.193,148.859
C02464=1241.026,-53.469,-37.479,-179.876,5.193,148.859
C02465=1241.020,-53.219,-37.491,-179.874,5.192,148.858
C02466=1241.015,-52.970,-37.504,-179.871,5.193,148.857
C02467=1241.010,-52.721,-37.516,-179.869,5.193,148.856
C02468=1241.006,-52.471,-37.529,-179.866,5.193,148.856
C02469=1241.001,-52.221,-37.542,-179.864,5.194,148.855
C02470=1240.995,-51.972,-37.554,-179.862,5.193,148.854
C02471=1240.990,-51.722,-37.566,-179.859,5.194,148.853
C02472=1240.985,-51.472,-37.579,-179.857,5.193,148.853
C02473=1240.980,-51.223,-37.592,-179.854,5.194,148.852
C02474=1240.974,-50.973,-37.605,-179.852,5.194,148.851
C02475=1240.970,-50.723,-37.618,-179.850,5.194,148.851
C02476=1240.965,-50.474,-37.631,-179.847,5.193,148.850
C02477=1240.960,-50.224,-37.643,-179.844,5.194,148.849
C02478=1240.955,-49.975,-37.656,-179.842,5.194,148.848
C02479=1240.950,-49.724,-37.668,-179.840,5.194,148.848
C02480=1240.944,-49.475,-37.681,-179.837,5.194,148.847
C02481=1240.939,-49.226,-37.694,-179.835,5.194,148.846
C02482=1240.934,-48.976,-37.706,-179.832,5.195,148.846
C02483=1240.929,-48.726,-37.719,-179.830,5.195,148.845
C02484=1240.923,-48.457,-37.733,-179.827,5.195,148.844
C02485=1240.918,-48.187,-37.747,-179.825,5.194,148.843
C02486=1240.913,-47.917,-37.761,-179.822,5.195,148.842
C02487=1240.906,-47.648,-37.775,-179.819,5.195,148.842
C02488=1240.902,-47.398,-37.788,-179.817,5.195,148.841
C02489=1240.897,-47.149,-37.800,-179.814,5.195,148.840
C02490=1240.892,-46.899,-37.813,-179.812,5.195,148.839
C02491=1240.886,-46.649,-37.826,-179.809,5.195,148.839
C02492=1240.881,-46.400,-37.839,-179.807,5.195,148.838
C02493=1240.876,-46.150,-37.852,-179.805,5.195,148.837
C02494=1240.872,-45.900,-37.865,-179.802,5.196,148.837
C02495=1240.866,-45.651,-37.878,-179.800,5.196,148.836
C02496=1240.861,-45.402,-37.890,-179.797,5.196,148.835
C02497=1240.856,-45.151,-37.903,-179.795,5.196,148.834
C02498=1240.851,-44.902,-37.916,-179.792,5.196,148.834
C02499=1240.845,-44.653,-37.929,-179.790,5.196,148.833
C02500=1240.841,-44.403,-37.942,-179.787,5.196,148.832
C02501=1240.835,-44.153,-37.955,-179.785,5.196,148.831
C02502=1240.830,-43.904,-37.967,-179.783,5.196,148.831
C02503=1240.825,-43.654,-37.981,-179.780,5.196,148.830
C02504=1240.820,-43.404,-37.993,-179.778,5.197,148.829
C02505=1240.816,-43.155,-38.007,-179.775,5.197,148.829
C02506=1240.810,-42.905,-38.020,-179.773,5.196,148.828
C02507=1240.805,-42.656,-38.033,-179.770,5.197,148.827
C02508=1240.800,-42.406,-38.046,-179.768,5.197,148.826
C02509=1240.795,-42.157,-38.058,-179.765,5.197,148.826
C02510=1240.789,-41.907,-38.072,-179.763,5.197,148.825
C02511=1240.785,-41.657,-38.085,-179.760,5.197,148.824
C02512=1240.780,-41.408,-38.097,-179.758,5.197,148.824
C02513=1240.775,-41.158,-38.112,-179.756,5.197,148.823
C02514=1240.770,-40.909,-38.124,-179.753,5.198,148.822
C02515=1240.764,-40.659,-38.137,-179.751,5.198,148.821
C02516=1240.759,-40.409,-38.150,-179.748,5.198,148.820
C02517=1240.754,-40.160,-38.163,-179.746,5.198,148.820
C02518=1240.749,-39.909,-38.176,-179.743,5.198,148.819
C02519=1240.744,-39.661,-38.190,-179.741,5.198,148.818
C02520=1240.739,-39.411,-38.202,-179.738,5.198,148.818
C02521=1240.734,-39.161,-38.216,-179.736,5.199,148.817
C02522=1240.728,-38.912,-38.229,-179.733,5.198,148.816
C02523=1240.724,-38.662,-38.241,-179.731,5.199,148.816
C02524=1240.718,-38.413,-38.255,-179.729,5.199,148.815
C02525=1240.714,-38.163,-38.268,-179.726,5.199,148.814
C02526=1240.708,-37.913,-38.282,-179.724,5.199,148.813
C02527=1240.703,-37.664,-38.294,-179.721,5.199,148.813
C02528=1240.699,-37.414,-38.308,-179.719,5.199,148.812
C02529=1240.693,-37.165,-38.321,-179.716,5.199,148.811
C02530=1240.688,-36.915,-38.334,-179.713,5.200,148.810
C02531=1240.682,-36.665,-38.347,-179.711,5.199,148.810
C02532=1240.678,-36.416,-38.361,-179.709,5.200,148.809
C02533=1240.672,-36.166,-38.374,-179.707,5.200,148.808
C02534=1240.668,-35.916,-38.387,-179.704,5.200,148.808
C02535=1240.663,-35.667,-38.400,-179.702,5.200,148.807
C02536=1240.658,-35.417,-38.414,-179.699,5.200,148.806
C02537=1240.653,-35.168,-38.427,-179.696,5.200,148.805
C02538=1240.648,-34.918,-38.441,-179.694,5.200,148.805
C02539=1240.642,-34.669,-38.453,-179.691,5.201,148.804
C02540=1240.637,-34.419,-38.467,-179.689,5.200,148.803
C02541=1240.632,-34.169,-38.480,-179.686,5.201,148.803
C02542=1240.627,-33.920,-38.493,-179.684,5.201,148.802
C02543=1240.622,-33.670,-38.506,-179.682,5.201,148.801
C02544=1240.616,-33.421,-38.520,-179.679,5.202,148.800
C02545=1240.612,-33.171,-38.533,-179.677,5.201,148.800
C02546=1240.606,-32.921,-38.547,-179.674,5.202,148.799
C02547=1240.602,-32.672,-38.560,-179.672,5.201,148.798
C02548=1240.596,-32.422,-38.573,-179.669,5.202,148.797
C02549=1240.592,-32.173,-38.587,-179.667,5.201,148.797
C02550=1240.587,-31.922,-38.601,-179.664,5.202,148.796
C02551=1240.581,-31.673,-38.613,-179.662,5.202,148.795
C02552=1240.576,-31.423,-38.628,-179.660,5.202,148.795
C02553=1240.571,-31.174,-38.640,-179.657,5.203,148.794
C02554=1240.566,-30.924,-38.654,-179.655,5.202,148.793
C02555=1240.561,-30.675,-38.668,-179.652,5.203,148.793
C02556=1240.556,-30.425,-38.681,-179.650,5.203,148.792
C02557=1240.550,-30.176,-38.694,-179.647,5.203,148.791
C02558=1240.546,-29.926,-38.708,-179.644,5.203,148.790
C02559=1240.540,-29.677,-38.721,-179.642,5.203,148.789
C02560=1240.536,-29.427,-38.735,-179.640,5.203,148.789
C02561=1240.530,-29.178,-38.748,-179.637,5.203,148.788
C02562=1240.525,-28.928,-38.762,-179.635,5.204,148.787
C02563=1240.521,-28.678,-38.775,-179.632,5.204,148.787
C02564=1240.515,-28.429,-38.789,-179.630,5.204,148.786
C02565=1240.511,-28.179,-38.802,-179.627,5.204,148.785
C02566=1240.505,-27.930,-38.816,-179.625,5.204,148.785
C02567=1240.500,-27.680,-38.830,-179.622,5.204,148.784
C02568=1240.495,-27.431,-38.843,-179.619,5.205,148.783
C02569=1240.490,-27.181,-38.857,-179.617,5.204,148.782
C02570=1240.486,-26.931,-38.870,-179.615,5.205,148.782
C02571=1240.480,-26.682,-38.884,-179.613,5.205,148.781
C02572=1240.475,-26.432,-38.898,-179.610,5.205,148.780
C02573=1240.470,-26.183,-38.911,-179.607,5.206,148.780
C02574=1240.465,-25.933,-38.925,-179.605,5.205,148.779
C02575=1240.460,-25.683,-38.939,-179.603,5.206,148.778
C02576=1240.455,-25.434,-38.952,-179.601,5.205,148.777
C02577=1240.450,-25.184,-38.966,-179.598,5.206,148.777
C02578=1240.445,-24.934,-38.980,-179.595,5.206,148.776
C02579=1240.440,-24.685,-38.993,-179.593,5.206,148.775
C02580=1240.435,-24.435,-39.007,-179.590,5.206,148.774
C02581=1240.429,-24.186,-39.021,-179.588,5.206,148.774
C02582=1240.425,-23.936,-39.034,-179.585,5.207,148.773
C02583=1240.420,-23.687,-39.048,-179.583,5.206,148.772
C02584=1240.414,-23.438,-39.062,-179.580,5.207,148.772
C02585=1240.409,-23.187,-39.076,-179.578,5.207,148.771
C02586=1240.405,-22.938,-39.089,-179.576,5.207,148.770
C02587=1240.399,-22.689,-39.103,-179.573,5.208,148.770
C02588=1240.394,-22.419,-39.118,-179.570,5.208,148.769
C02589=1240.388,-22.150,-39.133,-179.568,5.207,148.768
C02590=1240.383,-21.881,-39.148,-179.565,5.208,148.767
C02591=1240.377,-21.612,-39.162,-179.562,5.208,148.766
C02592=1240.372,-21.362,-39.177,-179.560,5.208,148.766
C02593=1240.367,-21.112,-39.190,-179.557,5.208,148.765
C02594=1240.362,-20.863,-39.204,-179.555,5.209,148.764
C02595=1240.357,-20.614,-39.218,-179.553,5.209,148.763
C02596=1240.352,-20.364,-39.232,-179.550,5.209,148.763
C02597=1240.347,-20.114,-39.245,-179.548,5.209,148.762
C02598=1240.342,-19.865,-39.259,-179.545,5.209,148.761
C02599=1240.337,-19.615,-39.274,-179.542,5.210,148.761
C02600=1240.333,-19.366,-39.287,-179.540,5.209,148.760
C02601=1240.327,-19.116,-39.301,-179.537,5.210,148.759
C02602=1240.322,-18.866,-39.315,-179.535,5.210,148.758
C02603=1240.317,-18.616,-39.329,-179.532,5.210,148.758
C02604=1240.311,-18.367,-39.343,-179.530,5.210,148.757
C02605=1240.307,-18.118,-39.357,-179.528,5.210,148.756
C02606=1240.302,-17.868,-39.371,-179.525,5.211,148.756
C02607=1240.296,-17.619,-39.384,-179.522,5.211,148.755
C02608=1240.291,-17.369,-39.399,-179.520,5.211,148.754
C02609=1240.286,-17.119,-39.413,-179.518,5.211,148.754
C02610=1240.281,-16.870,-39.427,-179.516,5.211,148.753
C02611=1240.276,-16.621,-39.440,-179.512,5.211,148.752
C02612=1240.272,-16.371,-39.455,-179.510,5.212,148.751
C02613=1240.267,-16.122,-39.469,-179.508,5.212,148.751
C02614=1240.261,-15.871,-39.482,-179.505,5.212,148.750
C02615=1240.256,-15.622,-39.496,-179.502,5.213,148.749
C02616=1240.251,-15.372,-39.511,-179.500,5.212,148.748
C02617=1240.246,-15.123,-39.525,-179.498,5.213,148.748
C02618=1240.241,-14.873,-39.539,-179.496,5.213,148.747
C02619=1240.236,-14.624,-39.553,-179.493,5.213,148.746
C02620=1240.231,-14.375,-39.567,-179.490,5.214,148.746
C02621=1240.226,-14.125,-39.581,-179.488,5.213,148.745
C02622=1240.221,-13.875,-39.595,-179.486,5.214,148.744
C02623=1240.216,-13.626,-39.609,-179.482,5.214,148.743
C02624=1240.211,-13.376,-39.624,-179.480,5.214,148.743
C02625=1240.206,-13.127,-39.638,-179.478,5.214,148.742
C02626=1240.201,-12.877,-39.652,-179.476,5.214,148.741
C02627=1240.196,-12.627,-39.666,-179.473,5.214,148.741
C02628=1240.190,-12.378,-39.680,-179.470,5.215,148.740
C02629=1240.185,-12.129,-39.695,-179.468,5.215,148.739
C02630=1240.180,-11.879,-39.709,-179.466,5.215,148.738
C02631=1240.175,-11.629,-39.723,-179.463,5.216,148.738
C02632=1240.170,-11.379,-39.737,-179.461,5.215,148.737
C02633=1240.165,-11.130,-39.751,-179.458,5.216,148.736
C02634=1240.161,-10.881,-39.765,-179.455,5.217,148.736
C02635=1240.156,-10.631,-39.779,-179.453,5.216,148.735
C02636=1240.151,-10.382,-39.794,-179.450,5.216,148.734
C02637=1240.146,-10.132,-39.808,-179.448,5.216,148.733
C02638=1240.140,-9.883,-39.822,-179.445,5.217,148.733
C02639=1240.135,-9.633,-39.836,-179.443,5.217,148.732
C02640=1240.130,-9.384,-39.850,-179.441,5.217,148.731
C02641=1240.125,-9.134,-39.865,-179.438,5.217,148.731
C02642=1240.120,-8.884,-39.879,-179.435,5.218,148.730
C02643=1240.116,-8.635,-39.894,-179.433,5.218,148.729
C02644=1240.110,-8.386,-39.908,-179.431,5.218,148.729
C02645=1240.105,-8.136,-39.923,-179.428,5.219,148.728
C02646=1240.100,-7.886,-39.937,-179.426,5.218,148.727
C02647=1240.095,-7.637,-39.951,-179.423,5.219,148.726
C02648=1240.090,-7.387,-39.965,-179.420,5.219,148.726
C02649=1240.085,-7.137,-39.980,-179.418,5.219,148.725
C02650=1240.080,-6.888,-39.995,-179.415,5.219,148.724
C02651=1240.075,-6.638,-40.009,-179.413,5.219,148.723
C02652=1240.070,-6.389,-40.023,-179.411,5.220,148.723
C02653=1240.065,-6.140,-40.037,-179.408,5.220,148.722
C02654=1240.060,-5.890,-40.051,-179.406,5.220,148.721
C02655=1240.055,-5.640,-40.066,-179.403,5.220,148.721
C02656=1240.050,-5.391,-40.081,-179.401,5.221,148.720
C02657=1240.045,-5.141,-40.095,-179.399,5.221,148.719
C02658=1240.040,-4.892,-40.109,-179.396,5.221,148.719
C02659=1240.035,-4.642,-40.124,-179.393,5.222,148.718
C02660=1240.030,-4.393,-40.139,-179.391,5.221,148.717
C02661=1240.024,-4.144,-40.153,-179.388,5.222,148.716
C02662=1240.019,-3.894,-40.167,-179.385,5.222,148.716
C02663=1240.014,-3.644,-40.182,-179.383,5.222,148.715
C02664=1240.010,-3.395,-40.197,-179.381,5.222,148.714
C02665=1240.005,-3.145,-40.211,-179.378,5.223,148.714
C02666=1240.000,-2.896,-40.225,-179.376,5.223,148.713
C02667=1239.995,-2.646,-40.239,-179.373,5.223,148.712
C02668=1239.989,-2.397,-40.255,-179.371,5.224,148.712
C02669=1239.984,-2.147,-40.269,-179.369,5.224,148.711
C02670=1239.980,-1.897,-40.284,-179.366,5.224,148.710
C02671=1239.975,-1.648,-40.299,-179.363,5.225,148.709
C02672=1239.970,-1.398,-40.313,-179.361,5.224,148.709
C02673=1239.965,-1.149,-40.327,-179.358,5.225,148.708
C02674=1239.960,-0.899,-40.343,-179.356,5.225,148.707
C02675=1239.955,-0.649,-40.357,-179.353,5.225,148.706
C02676=1239.949,-0.400,-40.371,-179.351,5.225,148.706
C02677=1239.944,-0.151,-40.386,-179.348,5.226,148.705
C02678=1239.939,0.098,-40.400,-179.346,5.226,148.704
C02679=1239.934,0.348,-40.416,-179.343,5.226,148.704
C02680=1239.929,0.597,-40.430,-179.341,5.227,148.703
C02681=1239.924,0.847,-40.444,-179.338,5.226,148.702
C02682=1239.920,1.096,-40.459,-179.336,5.227,148.702
C02683=1239.914,1.346,-40.474,-179.333,5.227,148.701
C02684=1239.909,1.595,-40.489,-179.331,5.227,148.700
C02685=1239.904,1.845,-40.503,-179.328,5.228,148.700
C02686=1239.899,2.095,-40.518,-179.326,5.228,148.699
C02687=1239.894,2.344,-40.533,-179.324,5.228,148.698
C02688=1239.889,2.594,-40.548,-179.321,5.228,148.697
C02689=1239.884,2.843,-40.563,-179.318,5.229,148.697
C02690=1239.879,3.093,-40.577,-179.316,5.229,148.696
C02691=1239.874,3.342,-40.592,-179.313,5.229,148.695
C02692=1239.869,3.611,-40.608,-179.311,5.229,148.695
C02693=1239.864,3.880,-40.624,-179.308,5.230,148.694
C02694=1239.858,4.149,-40.640,-179.305,5.231,148.693
C02695=1239.853,4.418,-40.656,-179.303,5.230,148.692
C02696=1239.848,4.667,-40.671,-179.300,5.230,148.692
C02697=1239.842,4.917,-40.686,-179.297,5.231,148.691
C02698=1239.838,5.166,-40.701,-179.295,5.231,148.690
C02699=1239.833,5.415,-40.715,-179.293,5.231,148.689
C02700=1239.827,5.665,-40.731,-179.290,5.232,148.689
C02701=1239.822,5.915,-40.745,-179.288,5.232,148.688
C02702=1239.818,6.164,-40.760,-179.285,5.232,148.687
C02703=1239.812,6.414,-40.775,-179.283,5.233,148.687
C02704=1239.808,6.664,-40.790,-179.280,5.233,148.686
C02705=1239.803,6.913,-40.805,-179.278,5.233,148.685
C02706=1239.798,7.163,-40.820,-179.275,5.233,148.685
C02707=1239.793,7.412,-40.835,-179.273,5.234,148.684
C02708=1239.787,7.662,-40.850,-179.270,5.234,148.683
C02709=1239.783,7.911,-40.865,-179.267,5.234,148.682
C02710=1239.778,8.160,-40.880,-179.265,5.234,148.682
C02711=1239.772,8.410,-40.895,-179.263,5.234,148.681
C02712=1239.768,8.659,-40.910,-179.260,5.235,148.680
C02713=1239.763,8.909,-40.924,-179.257,5.235,148.680
C02714=1239.757,9.158,-40.940,-179.255,5.235,148.679
C02715=1239.753,9.407,-40.955,-179.253,5.236,148.678
C02716=1239.748,9.658,-40.970,-179.250,5.236,148.678
C02717=1239.743,9.907,-40.985,-179.247,5.237,148.677
C02718=1239.738,10.156,-41.000,-179.245,5.236,148.676
C02719=1239.733,10.406,-41.015,-179.243,5.237,148.675
C02720=1239.728,10.655,-41.030,-179.240,5.237,148.675
C02721=1239.723,10.905,-41.045,-179.238,5.237,148.674
C02722=1239.718,11.154,-41.060,-179.235,5.238,148.673
C02723=1239.712,11.404,-41.075,-179.233,5.238,148.673
C02724=1239.708,11.653,-41.090,-179.230,5.239,148.672
C02725=1239.703,11.903,-41.106,-179.228,5.239,148.671
C02726=1239.698,12.152,-41.121,-179.225,5.239,148.671
C02727=1239.692,12.402,-41.136,-179.222,5.240,148.670
C02728=1239.688,12.651,-41.151,-179.220,5.239,148.669
C02729=1239.682,12.901,-41.166,-179.218,5.240,148.669
C02730=1239.678,13.150,-41.181,-179.215,5.240,148.668
C02731=1239.672,13.400,-41.196,-179.212,5.241,148.667
C02732=1239.668,13.649,-41.212,-179.210,5.240,148.666
C02733=1239.663,13.899,-41.227,-179.207,5.241,148.666
C02734=1239.658,14.148,-41.242,-179.205,5.242,148.665
C02735=1239.653,14.397,-41.258,-179.203,5.241,148.664
C02736=1239.648,14.647,-41.272,-179.200,5.242,148.664
C02737=1239.642,14.896,-41.288,-179.197,5.242,148.663
C02738=1239.638,15.146,-41.303,-179.195,5.243,148.662
C02739=1239.633,15.396,-41.319,-179.192,5.243,148.662
C02740=1239.628,15.645,-41.334,-179.190,5.243,148.661
C02741=1239.623,15.894,-41.349,-179.187,5.244,148.660
C02742=1239.618,16.143,-41.364,-179.185,5.244,148.659
C02743=1239.613,16.394,-41.380,-179.182,5.244,148.659
C02744=1239.608,16.643,-41.395,-179.180,5.245,148.658
C02745=1239.603,16.892,-41.410,-179.177,5.245,148.657
C02746=1239.598,17.142,-41.426,-179.175,5.245,148.657
C02747=1239.593,17.391,-41.441,-179.172,5.245,148.656
C02748=1239.588,17.641,-41.457,-179.170,5.246,148.655
C02749=1239.584,17.890,-41.472,-179.167,5.247,148.655
C02750=1239.578,18.140,-41.487,-179.165,5.246,148.654
C02751=1239.573,18.389,-41.503,-179.162,5.247,148.653
C02752=1239.569,18.639,-41.518,-179.160,5.247,148.653
C02753=1239.563,18.888,-41.534,-179.158,5.247,148.652
C02754=1239.558,19.138,-41.549,-179.155,5.248,148.651
C02755=1239.553,19.387,-41.564,-179.152,5.248,148.651
C02756=1239.549,19.637,-41.580,-179.150,5.249,148.650
C02757=1239.544,19.886,-41.595,-179.148,5.249,148.649
C02758=1239.538,20.135,-41.611,-179.145,5.249,148.649
C02759=1239.533,20.385,-41.626,-179.142,5.249,148.648
C02760=1239.529,20.634,-41.642,-179.139,5.250,148.647
C02761=1239.524,20.884,-41.657,-179.137,5.250,148.646
C02762=1239.518,21.133,-41.673,-179.135,5.250,148.646
C02763=1239.514,21.382,-41.688,-179.132,5.251,148.645
C02764=1239.509,21.632,-41.704,-179.129,5.251,148.644
C02765=1239.503,21.882,-41.720,-179.127,5.251,148.644
C02766=1239.499,22.131,-41.735,-179.125,5.252,148.643
C02767=1239.493,22.380,-41.750,-179.122,5.252,148.642
C02768=1239.489,22.630,-41.766,-179.119,5.253,148.642
C02769=1239.483,22.880,-41.782,-179.117,5.252,148.641
C02770=1239.479,23.129,-41.797,-179.115,5.253,148.640
C02771=1239.474,23.379,-41.813,-179.112,5.254,148.639
C02772=1239.468,23.628,-41.828,-179.109,5.254,148.639
C02773=1239.464,23.878,-41.843,-179.107,5.254,148.638
C02774=1239.459,24.128,-41.859,-179.104,5.254,148.637
C02775=1239.454,24.376,-41.875,-179.102,5.255,148.637
C02776=1239.449,24.626,-41.891,-179.099,5.256,148.636
C02777=1239.444,24.875,-41.906,-179.097,5.255,148.635
C02778=1239.439,25.125,-41.922,-179.094,5.256,148.635
C02779=1239.434,25.374,-41.938,-179.092,5.256,148.634
C02780=1239.428,25.624,-41.953,-179.089,5.257,148.633
C02781=1239.425,25.873,-41.969,-179.087,5.257,148.633
C02782=1239.419,26.122,-41.985,-179.084,5.257,148.632
C02783=1239.414,26.372,-42.000,-179.082,5.258,148.631
C02784=1239.409,26.622,-42.016,-179.079,5.258,148.631
C02785=1239.404,26.871,-42.032,-179.077,5.258,148.630
C02786=1239.400,27.120,-42.048,-179.074,5.259,148.629
C02787=1239.394,27.370,-42.064,-179.072,5.259,148.629
C02788=1239.389,27.619,-42.079,-179.069,5.260,148.628
C02789=1239.384,27.869,-42.095,-179.067,5.260,148.627
C02790=1239.379,28.119,-42.111,-179.064,5.260,148.627
C02791=1239.375,28.367,-42.126,-179.062,5.261,148.626
C02792=1239.370,28.617,-42.142,-179.059,5.261,148.625
C02793=1239.364,28.867,-42.158,-179.057,5.262,148.624
C02794=1239.359,29.116,-42.174,-179.054,5.262,148.624
C02795=1239.355,29.366,-42.190,-179.052,5.262,148.623
C02796=1239.349,29.634,-42.207,-179.049,5.263,148.622
C02797=1239.343,29.903,-42.224,-179.046,5.263,148.622
C02798=1239.338,30.172,-42.242,-179.043,5.263,148.621
C02799=1239.334,30.440,-42.258,-179.041,5.264,148.620
C02800=1239.328,30.689,-42.274,-179.039,5.264,148.619
C02801=1239.324,30.939,-42.290,-179.036,5.264,148.619
C02802=1239.318,31.188,-42.306,-179.033,5.265,148.618
C02803=1239.313,31.438,-42.321,-179.031,5.265,148.617
C02804=1239.309,31.687,-42.338,-179.028,5.266,148.617
C02805=1239.303,31.937,-42.354,-179.026,5.266,148.616
C02806=1239.299,32.186,-42.370,-179.023,5.266,148.615
C02807=1239.293,32.435,-42.386,-179.021,5.267,148.615
C02808=1239.288,32.686,-42.402,-179.018,5.267,148.614
C02809=1239.284,32.934,-42.418,-179.015,5.268,148.613
C02810=1239.279,33.183,-42.433,-179.013,5.268,148.613
C02811=1239.274,33.433,-42.450,-179.011,5.268,148.612
C02812=1239.269,33.682,-42.466,-179.008,5.269,148.611
C02813=1239.264,33.932,-42.481,-179.005,5.269,148.611
C02814=1239.259,34.181,-42.498,-179.003,5.269,148.610
C02815=1239.254,34.431,-42.514,-179.001,5.270,148.609
C02816=1239.249,34.680,-42.530,-178.998,5.270,148.609
C02817=1239.244,34.930,-42.546,-178.995,5.271,148.608
C02818=1239.239,35.179,-42.562,-178.993,5.271,148.607
C02819=1239.235,35.429,-42.578,-178.991,5.271,148.607
C02820=1239.229,35.678,-42.595,-178.988,5.272,148.606
C02821=1239.224,35.927,-42.610,-178.985,5.272,148.605
C02822=1239.220,36.177,-42.627,-178.983,5.273,148.605
C02823=1239.214,36.426,-42.642,-178.980,5.274,148.604
C02824=1239.210,36.676,-42.659,-178.978,5.273,148.603
C02825=1239.204,36.925,-42.675,-178.975,5.274,148.603
C02826=1239.200,37.175,-42.691,-178.973,5.274,148.602
C02827=1239.194,37.424,-42.707,-178.970,5.275,148.601
C02828=1239.190,37.673,-42.724,-178.968,5.276,148.601
C02829=1239.185,37.923,-42.739,-178.965,5.275,148.600
C02830=1239.180,38.172,-42.756,-178.963,5.276,148.599
C02831=1239.175,38.422,-42.771,-178.960,5.276,148.599
C02832=1239.170,38.671,-42.788,-178.958,5.277,148.598
C02833=1239.164,38.920,-42.805,-178.955,5.278,148.597
C02834=1239.160,39.170,-42.821,-178.953,5.277,148.596
C02835=1239.155,39.420,-42.838,-178.950,5.278,148.596
C02836=1239.150,39.669,-42.853,-178.948,5.278,148.595
C02837=1239.145,39.919,-42.870,-178.945,5.279,148.595
C02838=1239.140,40.168,-42.886,-178.943,5.280,148.594
C02839=1239.135,40.418,-42.902,-178.940,5.281,148.593
C02840=1239.130,40.666,-42.918,-178.938,5.280,148.593
C02841=1239.126,40.916,-42.935,-178.935,5.281,148.592
C02842=1239.120,41.165,-42.951,-178.933,5.281,148.591
C02843=1239.116,41.415,-42.967,-178.930,5.282,148.591
C02844=1239.110,41.664,-42.984,-178.927,5.283,148.590
C02845=1239.105,41.914,-43.000,-178.925,5.282,148.589
C02846=1239.101,42.163,-43.017,-178.923,5.283,148.589
C02847=1239.096,42.412,-43.033,-178.920,5.284,148.588
C02848=1239.091,42.662,-43.049,-178.917,5.284,148.587
C02849=1239.086,42.911,-43.065,-178.915,5.285,148.587
C02850=1239.081,43.161,-43.082,-178.912,5.285,148.586
C02851=1239.076,43.410,-43.099,-178.910,5.285,148.585
C02852=1239.071,43.660,-43.115,-178.908,5.286,148.585
C02853=1239.066,43.909,-43.132,-178.905,5.286,148.584
C02854=1239.061,44.158,-43.148,-178.902,5.287,148.583
C02855=1239.057,44.408,-43.165,-178.900,5.287,148.583
C02856=1239.051,44.657,-43.181,-178.897,5.288,148.582
C02857=1239.046,44.907,-43.197,-178.895,5.288,148.581
C02858=1239.042,45.156,-43.214,-178.892,5.288,148.581
C02859=1239.037,45.405,-43.230,-178.890,5.289,148.580
C02860=1239.032,45.655,-43.247,-178.887,5.289,148.579
C02861=1239.027,45.905,-43.264,-178.884,5.290,148.579
C02862=1239.022,46.154,-43.280,-178.882,5.291,148.578
C02863=1239.017,46.403,-43.297,-178.880,5.290,148.577
C02864=1239.012,46.652,-43.313,-178.877,5.291,148.577
C02865=1239.007,46.902,-43.330,-178.875,5.292,148.576
C02866=1239.002,47.151,-43.347,-178.872,5.292,148.575
C02867=1238.997,47.400,-43.363,-178.870,5.293,148.575
C02868=1238.992,47.650,-43.379,-178.867,5.294,148.574
C02869=1238.987,47.900,-43.396,-178.865,5.293,148.573
C02870=1238.982,48.149,-43.413,-178.862,5.294,148.573
C02871=1238.978,48.398,-43.429,-178.860,5.294,148.572
C02872=1238.973,48.648,-43.446,-178.857,5.295,148.571
C02873=1238.967,48.897,-43.463,-178.854,5.296,148.571
C02874=1238.963,49.146,-43.480,-178.852,5.296,148.570
C02875=1238.958,49.396,-43.496,-178.849,5.297,148.569
C02876=1238.953,49.645,-43.513,-178.847,5.297,148.569
C02877=1238.948,49.894,-43.530,-178.844,5.297,148.568
C02878=1238.944,50.144,-43.546,-178.842,5.298,148.567
C02879=1238.938,50.393,-43.563,-178.839,5.298,148.567
C02880=1238.933,50.642,-43.580,-178.836,5.299,148.566
C02881=1238.929,50.892,-43.597,-178.834,5.299,148.565
C02882=1238.924,51.142,-43.614,-178.831,5.300,148.565
C02883=1238.919,51.390,-43.630,-178.830,5.300,148.564
C02884=1238.914,51.640,-43.647,-178.827,5.301,148.564
C02885=1238.909,51.890,-43.664,-178.824,5.301,148.563
C02886=1238.904,52.139,-43.681,-178.822,5.302,148.562
C02887=1238.899,52.388,-43.697,-178.819,5.302,148.562
C02888=1238.894,52.638,-43.714,-178.816,5.303,148.561
C02889=1238.890,52.887,-43.731,-178.814,5.304,148.560
C02890=1238.884,53.136,-43.748,-178.812,5.303,148.559
C02891=1238.879,53.386,-43.765,-178.809,5.304,148.559
C02892=1238.875,53.635,-43.781,-178.806,5.305,148.558
C02893=1238.870,53.885,-43.799,-178.804,5.305,148.557
C02894=1238.865,54.134,-43.815,-178.801,5.306,148.557
C02895=1238.859,54.384,-43.832,-178.799,5.306,148.556
C02896=1238.855,54.633,-43.849,-178.796,5.307,148.555
C02897=1238.850,54.883,-43.866,-178.794,5.308,148.555
C02898=1238.845,55.132,-43.882,-178.792,5.308,148.554
C02899=1238.840,55.381,-43.900,-178.789,5.308,148.554
C02900=1238.835,55.650,-43.919,-178.786,5.309,148.553
C02901=1238.830,55.917,-43.936,-178.783,5.309,148.552
C02902=1238.824,56.186,-43.955,-178.781,5.310,148.551
C02903=1238.819,56.454,-43.973,-178.778,5.310,148.551
C02904=1238.814,56.704,-43.990,-178.775,5.311,148.550
C02905=1238.809,56.953,-44.007,-178.773,5.311,148.549
C02906=1238.804,57.203,-44.024,-178.770,5.312,148.549
C02907=1238.800,57.453,-44.041,-178.767,5.313,148.548
C02908=1238.794,57.701,-44.058,-178.765,5.313,148.548
C02909=1238.790,57.951,-44.075,-178.763,5.314,148.547
C02910=1238.784,58.200,-44.092,-178.760,5.315,148.546
C02911=1238.780,58.450,-44.109,-178.757,5.315,148.546
C02912=1238.775,58.700,-44.126,-178.755,5.315,148.545
C02913=1238.770,58.948,-44.143,-178.753,5.316,148.544
C02914=1238.765,59.198,-44.160,-178.750,5.316,148.544
C02915=1238.760,59.447,-44.177,-178.747,5.317,148.543
C02916=1238.755,59.697,-44.194,-178.745,5.317,148.542
C02917=1238.751,59.946,-44.212,-178.742,5.318,148.542
C02918=1238.746,60.196,-44.229,-178.740,5.319,148.541
C02919=1238.740,60.445,-44.246,-178.737,5.319,148.541
C02920=1238.736,60.694,-44.263,-178.735,5.320,148.540
C02921=1238.730,60.943,-44.280,-178.733,5.320,148.539
C02922=1238.726,61.193,-44.297,-178.730,5.320,148.539
C02923=1238.721,61.442,-44.315,-178.727,5.321,148.538
C02924=1238.717,61.691,-44.332,-178.725,5.322,148.537
C02925=1238.711,61.941,-44.349,-178.722,5.322,148.537
C02926=1238.706,62.190,-44.367,-178.720,5.323,148.536
C02927=1238.701,62.439,-44.383,-178.717,5.323,148.535
C02928=1238.696,62.689,-44.401,-178.714,5.324,148.535
C02929=1238.692,62.938,-44.418,-178.712,5.325,148.534
C02930=1238.687,63.188,-44.435,-178.710,5.326,148.533
C02931=1238.682,63.438,-44.452,-178.707,5.326,148.533
C02932=1238.677,63.686,-44.470,-178.705,5.326,148.532
C02933=1238.672,63.936,-44.487,-178.702,5.326,148.531
C02934=1238.667,64.185,-44.505,-178.700,5.327,148.531
C02935=1238.662,64.434,-44.521,-178.697,5.328,148.530
C02936=1238.657,64.683,-44.539,-178.694,5.328,148.529
C02937=1238.652,64.933,-44.557,-178.692,5.329,148.529
C02938=1238.648,65.183,-44.573,-178.689,5.329,148.528
C02939=1238.643,65.432,-44.591,-178.687,5.330,148.528
C02940=1238.637,65.682,-44.609,-178.684,5.331,148.527
C02941=1238.633,65.930,-44.626,-178.682,5.332,148.526
C02942=1238.628,66.180,-44.643,-178.679,5.332,148.526
C02943=1238.623,66.429,-44.661,-178.676,5.333,148.525
C02944=1238.619,66.679,-44.678,-178.674,5.333,148.524
C02945=1238.614,66.928,-44.696,-178.672,5.333,148.524
C02946=1238.609,67.178,-44.713,-178.669,5.334,148.523
C02947=1238.604,67.426,-44.730,-178.667,5.335,148.523
C02948=1238.599,67.676,-44.747,-178.664,5.335,148.522
C02949=1238.594,67.925,-44.765,-178.662,5.336,148.521
C02950=1238.589,68.174,-44.783,-178.659,5.336,148.521
C02951=1238.584,68.424,-44.800,-178.656,5.337,148.520
C02952=1238.579,68.673,-44.818,-178.654,5.338,148.519
C02953=1238.574,68.923,-44.835,-178.651,5.338,148.519
C02954=1238.569,69.172,-44.853,-178.649,5.339,148.518
C02955=1238.565,69.421,-44.870,-178.646,5.340,148.518
C02956=1238.560,69.670,-44.888,-178.644,5.340,148.517
C02957=1238.555,69.920,-44.906,-178.641,5.341,148.516
C02958=1238.550,70.169,-44.923,-178.638,5.342,148.516
C02959=1238.545,70.418,-44.941,-178.636,5.342,148.515
C02960=1238.541,70.667,-44.959,-178.633,5.343,148.514
C02961=1238.535,70.917,-44.976,-178.631,5.343,148.514
C02962=1238.530,71.166,-44.994,-178.629,5.343,148.513
C02963=1238.525,71.416,-45.011,-178.626,5.344,148.513
C02964=1238.520,71.665,-45.029,-178.624,5.345,148.512
C02965=1238.516,71.914,-45.046,-178.621,5.345,148.511
C02966=1238.511,72.163,-45.064,-178.619,5.346,148.511
C02967=1238.506,72.413,-45.082,-178.616,5.347,148.510
C02968=1238.501,72.662,-45.100,-178.613,5.347,148.509
C02969=1238.496,72.912,-45.118,-178.611,5.348,148.509
C02970=1238.491,73.161,-45.135,-178.608,5.349,148.508
C02971=1238.487,73.410,-45.152,-178.606,5.349,148.507
C02972=1238.482,73.659,-45.170,-178.603,5.350,148.507
C02973=1238.477,73.909,-45.188,-178.601,5.350,148.506
C02974=1238.472,74.158,-45.205,-178.598,5.351,148.505
C02975=1238.467,74.408,-45.223,-178.595,5.352,148.505
C02976=1238.463,74.657,-45.242,-178.593,5.352,148.504
C02977=1238.458,74.907,-45.260,-178.591,5.353,148.504
C02978=1238.452,75.156,-45.277,-178.588,5.354,148.503
C02979=1238.448,75.405,-45.294,-178.585,5.354,148.502
C02980=1238.443,75.654,-45.312,-178.583,5.355,148.502
C02981=1238.438,75.904,-45.330,-178.580,5.356,148.501
C02982=1238.433,76.153,-45.348,-178.577,5.356,148.500
C02983=1238.428,76.403,-45.366,-178.575,5.357,148.500
C02984=1238.423,76.652,-45.384,-178.573,5.358,148.499
C02985=1238.418,76.901,-45.402,-178.570,5.358,148.499
C02986=1238.414,77.150,-45.420,-178.567,5.359,148.498
C02987=1238.409,77.399,-45.438,-178.565,5.359,148.497
C02988=1238.404,77.648,-45.456,-178.563,5.359,148.497
C02989=1238.399,77.898,-45.474,-178.560,5.360,148.496
C02990=1238.394,78.148,-45.492,-178.558,5.361,148.496
C02991=1238.389,78.397,-45.509,-178.555,5.362,148.495
C02992=1238.384,78.646,-45.527,-178.553,5.362,148.494
C02993=1238.379,78.896,-45.545,-178.550,5.363,148.494
C02994=1238.375,79.145,-45.563,-178.547,5.363,148.493
C02995=1238.370,79.394,-45.581,-178.545,5.364,148.492
C02996=1238.365,79.643,-45.599,-178.543,5.365,148.492
C02997=1238.360,79.892,-45.617,-178.540,5.366,148.491
C02998=1238.355,80.142,-45.635,-178.537,5.366,148.491
C02999=1238.351,80.391,-45.653,-178.535,5.367,148.490
C03000=1238.346,80.641,-45.671,-178.532,5.367,148.489
C03001=1238.341,80.890,-45.689,-178.530,5.368,148.489
C03002=1238.336,81.139,-45.707,-178.527,5.369,148.488
C03003=1238.331,81.388,-45.725,-178.525,5.370,148.488
C03004=1238.326,81.656,-45.745,-178.522,5.370,148.487
C03005=1238.321,81.925,-45.764,-178.519,5.372,148.486
C03006=1238.315,82.193,-45.784,-178.516,5.372,148.486
C03007=1238.310,82.462,-45.804,-178.514,5.373,148.485
C03008=1238.306,82.711,-45.822,-178.511,5.373,148.484
C03009=1238.301,82.961,-45.840,-178.509,5.374,148.484
C03010=1238.296,83.210,-45.858,-178.506,5.375,148.483
C03011=1238.291,83.459,-45.876,-178.503,5.375,148.482
C03012=1238.286,83.708,-45.894,-178.501,5.376,148.482
C03013=1238.282,83.958,-45.912,-178.499,5.377,148.481
C03014=1238.277,84.207,-45.930,-178.496,5.377,148.481
C03015=1238.271,84.457,-45.949,-178.493,5.378,148.480
C03016=1238.266,84.706,-45.967,-178.491,5.379,148.479
C03017=1238.261,84.955,-45.985,-178.489,5.380,148.479
C03018=1238.257,85.205,-46.003,-178.486,5.380,148.478
C03019=1238.252,85.453,-46.022,-178.483,5.381,148.478
C03020=1238.247,85.703,-46.040,-178.481,5.381,148.477
C03021=1238.242,85.952,-46.058,-178.478,5.382,148.476
C03022=1238.237,86.202,-46.077,-178.476,5.383,148.476
C03023=1238.232,86.451,-46.095,-178.473,5.384,148.475
C03024=1238.228,86.700,-46.112,-178.471,5.384,148.474
C03025=1238.223,86.949,-46.131,-178.468,5.385,148.474
C03026=1238.218,87.198,-46.149,-178.465,5.385,148.473
C03027=1238.214,87.448,-46.168,-178.463,5.386,148.473
C03028=1238.208,87.697,-46.186,-178.461,5.387,148.472
C03029=1238.204,87.946,-46.205,-178.458,5.388,148.471
C03030=1238.199,88.196,-46.223,-178.455,5.388,148.471
C03031=1238.194,88.445,-46.241,-178.453,5.389,148.470
C03032=1238.189,88.694,-46.259,-178.451,5.390,148.470
C03033=1238.184,88.944,-46.278,-178.448,5.390,148.469
C03034=1238.180,89.193,-46.297,-178.445,5.391,148.468
C03035=1238.175,89.442,-46.315,-178.443,5.392,148.468
C03036=1238.170,89.691,-46.333,-178.440,5.392,148.467
C03037=1238.165,89.940,-46.352,-178.438,5.393,148.467
C03038=1238.160,90.190,-46.370,-178.435,5.394,148.466
C03039=1238.155,90.439,-46.388,-178.432,5.395,148.465
C03040=1238.151,90.688,-46.407,-178.430,5.396,148.465
C03041=1238.146,90.938,-46.426,-178.428,5.397,148.464
C03042=1238.141,91.187,-46.444,-178.425,5.398,148.464
C03043=1238.136,91.436,-46.463,-178.422,5.398,148.463
C03044=1238.131,91.686,-46.482,-178.420,5.399,148.462
C03045=1238.126,91.935,-46.500,-178.417,5.399,148.462
C03046=1238.122,92.184,-46.518,-178.415,5.400,148.461
C03047=1238.117,92.433,-46.536,-178.412,5.401,148.461
C03048=1238.112,92.683,-46.555,-178.410,5.402,148.460
C03049=1238.107,92.931,-46.574,-178.407,5.402,148.459
C03050=1238.102,93.181,-46.592,-178.405,5.403,148.459
C03051=1238.097,93.430,-46.611,-178.402,5.404,148.458
C03052=1238.092,93.679,-46.629,-178.400,5.404,148.458
C03053=1238.088,93.929,-46.648,-178.397,5.405,148.457
C03054=1238.083,94.178,-46.667,-178.395,5.406,148.457
C03055=1238.078,94.427,-46.685,-178.392,5.407,148.456
C03056=1238.073,94.677,-46.705,-178.390,5.407,148.455
C03057=1238.068,94.926,-46.723,-178.387,5.408,148.455
C03058=1238.064,95.175,-46.741,-178.384,5.409,148.454
C03059=1238.059,95.425,-46.760,-178.382,5.410,148.454
C03060=1238.054,95.673,-46.779,-178.379,5.411,148.453
C03061=1238.049,95.923,-46.797,-178.377,5.411,148.452
C03062=1238.044,96.172,-46.817,-178.374,5.412,148.452
C03063=1238.039,96.421,-46.835,-178.372,5.413,148.451
C03064=1238.035,96.671,-46.854,-178.369,5.414,148.450
C03065=1238.030,96.920,-46.872,-178.367,5.414,148.450
C03066=1238.025,97.169,-46.891,-178.364,5.415,148.449
C03067=1238.020,97.419,-46.910,-178.362,5.416,148.449
C03068=1238.015,97.667,-46.929,-178.359,5.416,148.448
C03069=1238.011,97.917,-46.948,-178.357,5.417,148.447
C03070=1238.006,98.166,-46.966,-178.354,5.418,148.447
C03071=1238.000,98.415,-46.986,-178.352,5.419,148.446
C03072=1237.996,98.665,-47.004,-178.349,5.420,148.446
C03073=1237.991,98.914,-47.023,-178.346,5.421,148.445
C03074=1237.987,99.163,-47.042,-178.343,5.421,148.444
C03075=1237.981,99.412,-47.061,-178.341,5.422,148.444
C03076=1237.977,99.662,-47.080,-178.339,5.423,148.443
C03077=1237.972,99.911,-47.098,-178.336,5.424,148.443
C03078=1237.967,100.160,-47.117,-178.333,5.424,148.442
C03079=1237.962,100.409,-47.137,-178.331,5.425,148.442
C03080=1237.957,100.658,-47.155,-178.329,5.426,148.441
C03081=1237.953,100.908,-47.174,-178.326,5.426,148.440
C03082=1237.948,101.157,-47.193,-178.324,5.427,148.440
C03083=1237.943,101.407,-47.212,-178.321,5.429,148.439
C03084=1237.938,101.655,-47.231,-178.318,5.429,148.439
C03085=1237.934,101.905,-47.250,-178.316,5.430,148.438
C03086=1237.929,102.153,-47.269,-178.313,5.431,148.438
C03087=1237.924,102.404,-47.288,-178.311,5.432,148.437
C03088=1237.919,102.652,-47.307,-178.308,5.432,148.436
C03089=1237.915,102.902,-47.326,-178.306,5.433,148.436
C03090=1237.910,103.150,-47.345,-178.303,5.434,148.435
C03091=1237.905,103.401,-47.364,-178.301,5.435,148.435
C03092=1237.900,103.649,-47.383,-178.298,5.435,148.434
C03093=1237.896,103.899,-47.402,-178.296,5.437,148.434
C03094=1237.890,104.147,-47.422,-178.293,5.438,148.433
C03095=1237.886,104.397,-47.441,-178.290,5.438,148.432
C03096=1237.881,104.646,-47.459,-178.288,5.439,148.432
C03097=1237.876,104.896,-47.479,-178.286,5.440,148.431
C03098=1237.871,105.144,-47.498,-178.283,5.440,148.431
C03099=1237.866,105.394,-47.517,-178.280,5.441,148.430
C03100=1237.861,105.643,-47.537,-178.278,5.442,148.430
C03101=1237.857,105.893,-47.555,-178.276,5.443,148.429
C03102=1237.851,106.142,-47.574,-178.272,5.444,148.428
C03103=1237.847,106.391,-47.593,-178.270,5.445,148.428
C03104=1237.842,106.640,-47.613,-178.268,5.446,148.427
C03105=1237.837,106.889,-47.632,-178.265,5.446,148.427
C03106=1237.833,107.138,-47.651,-178.262,5.447,148.426
C03107=1237.828,107.387,-47.671,-178.260,5.448,148.425
C03108=1237.823,107.656,-47.692,-178.258,5.449,148.425
C03109=1237.817,107.925,-47.712,-178.255,5.450,148.424
C03110=1237.812,108.193,-47.733,-178.252,5.451,148.424
C03111=1237.807,108.461,-47.754,-178.249,5.451,148.423
C03112=1237.802,108.711,-47.773,-178.247,5.452,148.422
C03113=1237.798,108.960,-47.792,-178.244,5.454,148.422
C03114=1237.793,109.209,-47.812,-178.241,5.454,148.421
C03115=1237.788,109.458,-47.831,-178.239,5.455,148.421
C03116=1237.783,109.707,-47.850,-178.236,5.456,148.420
C03117=1237.779,109.957,-47.870,-178.234,5.457,148.420
C03118=1237.773,110.205,-47.889,-178.231,5.457,148.419
C03119=1237.769,110.455,-47.908,-178.229,5.458,148.418
C03120=1237.765,110.704,-47.928,-178.226,5.460,148.418
C03121=1237.759,110.953,-47.947,-178.224,5.460,148.417
C03122=1237.754,111.203,-47.966,-178.221,5.461,148.417
C03123=1237.750,111.452,-47.986,-178.219,5.462,148.416
C03124=1237.745,111.701,-48.005,-178.216,5.463,148.415
C03125=1237.740,111.950,-48.025,-178.214,5.463,148.415
C03126=1237.735,112.199,-48.044,-178.211,5.464,148.414
C03127=1237.730,112.449,-48.063,-178.208,5.466,148.414
C03128=1237.726,112.698,-48.083,-178.206,5.466,148.413
C03129=1237.721,112.947,-48.102,-178.204,5.467,148.413
C03130=1237.716,113.196,-48.122,-178.201,5.468,148.412
C03131=1237.712,113.445,-48.142,-178.198,5.468,148.411
C03132=1237.706,113.694,-48.161,-178.196,5.469,148.411
C03133=1237.702,113.944,-48.181,-178.193,5.471,148.410
C03134=1237.697,114.193,-48.200,-178.190,5.472,148.410
C03135=1237.692,114.442,-48.219,-178.188,5.473,148.409
C03136=1237.688,114.692,-48.239,-178.186,5.473,148.409
C03137=1237.683,114.941,-48.259,-178.183,5.474,148.408
C03138=1237.678,115.189,-48.278,-178.181,5.475,148.408
C03139=1237.673,115.439,-48.298,-178.178,5.476,148.407
C03140=1237.668,115.689,-48.318,-178.175,5.477,148.406
C03141=1237.663,115.937,-48.337,-178.173,5.478,148.406
C03142=1237.659,116.186,-48.357,-178.170,5.479,148.405
C03143=1237.655,116.436,-48.376,-178.168,5.479,148.405
C03144=1237.649,116.684,-48.396,-178.166,5.480,148.404
C03145=1237.644,116.934,-48.415,-178.163,5.482,148.404
C03146=1237.640,117.183,-48.436,-178.160,5.482,148.403
C03147=1237.635,117.433,-48.455,-178.158,5.483,148.403
C03148=1237.630,117.681,-48.475,-178.155,5.484,148.402
C03149=1237.625,117.931,-48.494,-178.153,5.484,148.401
C03150=1237.621,118.180,-48.515,-178.150,5.486,148.401
C03151=1237.615,118.429,-48.534,-178.147,5.487,148.400
C03152=1237.611,118.678,-48.554,-178.145,5.488,148.400
C03153=1237.606,118.927,-48.574,-178.143,5.489,148.399
C03154=1237.601,119.177,-48.594,-178.140,5.489,148.399
C03155=1237.596,119.426,-48.613,-178.137,5.490,148.398
C03156=1237.592,119.675,-48.633,-178.135,5.492,148.398
C03157=1237.587,119.924,-48.653,-178.132,5.492,148.397
C03158=1237.582,120.174,-48.673,-178.130,5.493,148.397
C03159=1237.577,120.422,-48.693,-178.127,5.494,148.396
C03160=1237.572,120.672,-48.712,-178.125,5.495,148.395
C03161=1237.568,120.921,-48.733,-178.122,5.496,148.395
C03162=1237.563,121.170,-48.752,-178.120,5.497,148.394
C03163=1237.558,121.419,-48.772,-178.117,5.498,148.394
C03164=1237.553,121.668,-48.792,-178.115,5.499,148.393
C03165=1237.549,121.918,-48.812,-178.112,5.499,148.393
C03166=1237.544,122.167,-48.832,-178.109,5.501,148.392
C03167=1237.540,122.416,-48.852,-178.107,5.502,148.392
C03168=1237.534,122.664,-48.872,-178.104,5.502,148.391
C03169=1237.530,122.914,-48.891,-178.102,5.503,148.391
C03170=1237.525,123.163,-48.911,-178.100,5.504,148.390
C03171=1237.521,123.412,-48.931,-178.096,5.505,148.389
C03172=1237.516,123.662,-48.951,-178.094,5.506,148.389
C03173=1237.511,123.910,-48.971,-178.092,5.507,148.388
C03174=1237.506,124.160,-48.991,-178.089,5.508,148.388
C03175=1237.502,124.409,-49.011,-178.086,5.510,148.387
C03176=1237.496,124.658,-49.032,-178.084,5.510,148.387
C03177=1237.492,124.908,-49.052,-178.082,5.511,148.386
C03178=1237.487,125.157,-49.072,-178.079,5.512,148.385
C03179=1237.482,125.405,-49.091,-178.076,5.512,148.385
C03180=1237.477,125.654,-49.112,-178.074,5.514,148.384
C03181=1237.473,125.904,-49.131,-178.071,5.515,148.384
C03182=1237.468,126.153,-49.152,-178.069,5.516,148.383
C03183=1237.464,126.402,-49.171,-178.066,5.517,148.383
C03184=1237.458,126.652,-49.192,-178.063,5.518,148.382
C03185=1237.454,126.901,-49.213,-178.061,5.519,148.382
C03186=1237.449,127.149,-49.232,-178.059,5.520,148.381
C03187=1237.444,127.398,-49.252,-178.056,5.521,148.381
C03188=1237.440,127.647,-49.273,-178.054,5.521,148.380
C03189=1237.435,127.897,-49.293,-178.051,5.523,148.379
C03190=1237.430,128.146,-49.313,-178.049,5.524,148.379
C03191=1237.425,128.395,-49.334,-178.046,5.524,148.378
C03192=1237.421,128.645,-49.354,-178.044,5.525,148.378
C03193=1237.416,128.894,-49.374,-178.041,5.527,148.377
C03194=1237.411,129.142,-49.394,-178.038,5.527,148.377
C03195=1237.406,129.392,-49.414,-178.036,5.528,148.376
C03196=1237.401,129.641,-49.435,-178.033,5.529,148.376
C03197=1237.397,129.890,-49.455,-178.031,5.531,148.375
C03198=1237.392,130.139,-49.475,-178.028,5.532,148.375
C03199=1237.387,130.389,-49.496,-178.026,5.532,148.374
C03200=1237.382,130.637,-49.516,-178.023,5.533,148.374
C03201=1237.378,130.886,-49.536,-178.020,5.535,148.373
C03202=1237.373,131.136,-49.556,-178.018,5.536,148.373
C03203=1237.368,131.385,-49.577,-178.016,5.536,148.372
C03204=1237.364,131.634,-49.597,-178.013,5.537,148.372
C03205=1237.359,131.883,-49.618,-178.010,5.539,148.371
C03206=1237.355,132.132,-49.638,-178.008,5.539,148.370
C03207=1237.349,132.382,-49.658,-178.006,5.540,148.370
C03208=1237.344,132.630,-49.678,-178.003,5.541,148.369
C03209=1237.340,132.879,-49.699,-178.000,5.543,148.369
C03210=1237.335,133.128,-49.720,-177.998,5.544,148.368
C03211=1237.330,133.377,-49.740,-177.996,5.545,148.368
C03212=1237.325,133.647,-49.762,-177.992,5.546,148.367
C03213=1237.321,133.915,-49.784,-177.990,5.547,148.367
C03214=1237.315,134.183,-49.806,-177.987,5.548,148.366
C03215=1237.310,134.452,-49.828,-177.984,5.549,148.365
C03216=1237.305,134.701,-49.848,-177.982,5.550,148.365
C03217=1237.300,134.951,-49.869,-177.979,5.551,148.364
C03218=1237.295,135.200,-49.890,-177.977,5.552,148.364
C03219=1237.291,135.448,-49.910,-177.974,5.553,148.363
C03220=1237.286,135.698,-49.931,-177.972,5.554,148.363
C03221=1237.281,135.947,-49.951,-177.969,5.555,148.362
C03222=1237.276,136.196,-49.972,-177.967,5.556,148.362
C03223=1237.272,136.445,-49.993,-177.964,5.557,148.361
C03224=1237.268,136.695,-50.013,-177.961,5.558,148.361
C03225=1237.263,136.944,-50.034,-177.959,5.559,148.360
C03226=1237.258,137.193,-50.055,-177.956,5.560,148.360
C03227=1237.253,137.442,-50.076,-177.954,5.561,148.359
C03228=1237.249,137.691,-50.096,-177.951,5.563,148.359
C03229=1237.244,137.940,-50.117,-177.949,5.564,148.358
C03230=1237.239,138.189,-50.137,-177.946,5.564,148.358
C03231=1237.235,138.438,-50.158,-177.944,5.566,148.357
C03232=1237.230,138.687,-50.179,-177.941,5.567,148.357
C03233=1237.225,138.936,-50.199,-177.939,5.568,148.356
C03234=1237.220,139.186,-50.220,-177.936,5.569,148.356
C03235=1237.215,139.435,-50.240,-177.933,5.570,148.355
C03236=1237.210,139.684,-50.261,-177.931,5.571,148.355
C03237=1237.206,139.933,-50.282,-177.928,5.571,148.354
C03238=1237.201,140.182,-50.303,-177.926,5.573,148.354
C03239=1237.196,140.431,-50.323,-177.923,5.574,148.353
C03240=1237.191,140.680,-50.344,-177.921,5.575,148.353
C03241=1237.187,140.929,-50.365,-177.918,5.576,148.352
C03242=1237.182,141.179,-50.387,-177.916,5.577,148.352
C03243=1237.178,141.427,-50.407,-177.913,5.578,148.351
C03244=1237.173,141.677,-50.428,-177.910,5.580,148.351
C03245=1237.168,141.926,-50.448,-177.908,5.581,148.350
C03246=1237.163,142.175,-50.469,-177.906,5.582,148.350
C03247=1237.159,142.423,-50.490,-177.903,5.583,148.349
C03248=1237.154,142.673,-50.511,-177.901,5.584,148.349
C03249=1237.149,142.922,-50.532,-177.898,5.585,148.348
C03250=1237.144,143.171,-50.553,-177.895,5.587,148.348
C03251=1237.140,143.421,-50.574,-177.893,5.587,148.347
C03252=1237.136,143.669,-50.595,-177.891,5.588,148.347
C03253=1237.130,143.918,-50.616,-177.887,5.590,148.346
C03254=1237.125,144.168,-50.637,-177.885,5.590,148.345
C03255=1237.121,144.417,-50.657,-177.883,5.591,148.345
C03256=1237.116,144.665,-50.679,-177.880,5.593,148.344
C03257=1237.111,144.914,-50.699,-177.877,5.594,148.344
C03258=1237.107,145.164,-50.721,-177.875,5.594,148.343
C03259=1237.102,145.413,-50.742,-177.872,5.596,148.343
C03260=1237.098,145.662,-50.763,-177.870,5.597,148.342
C03261=1237.092,145.911,-50.784,-177.867,5.598,148.342
C03262=1237.088,146.160,-50.804,-177.864,5.599,148.341
C03263=1237.083,146.408,-50.826,-177.862,5.600,148.341
C03264=1237.079,146.658,-50.847,-177.860,5.601,148.340
C03265=1237.074,146.907,-50.867,-177.857,5.603,148.340
C03266=1237.069,147.156,-50.889,-177.854,5.604,148.339
C03267=1237.064,147.405,-50.910,-177.852,5.605,148.339
C03268=1237.060,147.654,-50.931,-177.849,5.606,148.338
C03269=1237.055,147.904,-50.953,-177.847,5.607,148.338
C03270=1237.050,148.153,-50.974,-177.845,5.608,148.337
C03271=1237.045,148.401,-50.995,-177.842,5.610,148.337
C03272=1237.041,148.650,-51.016,-177.840,5.611,148.336
C03273=1237.036,148.899,-51.037,-177.837,5.611,148.336
C03274=1237.031,149.149,-51.059,-177.834,5.613,148.335
C03275=1237.027,149.397,-51.080,-177.832,5.614,148.335
C03276=1237.022,149.647,-51.101,-177.829,5.616,148.334
C03277=1237.017,149.896,-51.122,-177.827,5.616,148.334
C03278=1237.013,150.145,-51.144,-177.824,5.617,148.333
C03279=1237.008,150.394,-51.164,-177.821,5.619,148.333
C03280=1237.003,150.643,-51.186,-177.819,5.620,148.332
C03281=1236.998,150.892,-51.207,-177.817,5.620,148.332
C03282=1236.993,151.141,-51.228,-177.814,5.622,148.331
C03283=1236.989,151.391,-51.250,-177.811,5.623,148.331
C03284=1236.985,151.639,-51.271,-177.809,5.624,148.330
C03285=1236.980,151.888,-51.292,-177.806,5.625,148.330
C03286=1236.975,152.138,-51.314,-177.804,5.626,148.329
C03287=1236.970,152.386,-51.335,-177.801,5.628,148.329
C03288=1236.965,152.636,-51.356,-177.799,5.629,148.328
C03289=1236.961,152.884,-51.378,-177.796,5.630,148.328
C03290=1236.956,153.134,-51.399,-177.793,5.631,148.327
C03291=1236.952,153.382,-51.421,-177.791,5.632,148.327
C03292=1236.947,153.631,-51.442,-177.788,5.634,148.326
C03293=1236.942,153.881,-51.464,-177.786,5.635,148.326
C03294=1236.937,154.130,-51.485,-177.784,5.636,148.325
C03295=1236.933,154.379,-51.506,-177.781,5.637,148.325
C03296=1236.928,154.627,-51.527,-177.778,5.638,148.324
C03297=1236.924,154.877,-51.549,-177.776,5.639,148.324
C03298=1236.918,155.126,-51.570,-177.773,5.641,148.323
C03299=1236.914,155.375,-51.592,-177.771,5.642,148.323
C03300=1236.909,155.624,-51.614,-177.768,5.643,148.322
C03301=1236.904,155.872,-51.636,-177.766,5.644,148.322
C03302=1236.899,156.122,-51.657,-177.764,5.645,148.322
C03303=1236.895,156.371,-51.679,-177.760,5.647,148.321
C03304=1236.890,156.620,-51.700,-177.758,5.648,148.321
C03305=1236.886,156.869,-51.721,-177.755,5.649,148.320
C03306=1236.881,157.118,-51.743,-177.753,5.650,148.320
C03307=1236.877,157.367,-51.765,-177.750,5.651,148.319
C03308=1236.872,157.615,-51.786,-177.748,5.653,148.319
C03309=1236.867,157.865,-51.808,-177.746,5.654,148.318
C03310=1236.862,158.114,-51.829,-177.743,5.655,148.318
C03311=1236.858,158.363,-51.851,-177.740,5.656,148.317
C03312=1236.853,158.612,-51.873,-177.737,5.658,148.317
C03313=1236.848,158.861,-51.895,-177.735,5.659,148.316
C03314=1236.844,159.110,-51.916,-177.733,5.659,148.316
C03315=1236.839,159.359,-51.938,-177.730,5.661,148.315
C03316=1236.834,159.628,-51.962,-177.727,5.662,148.315
C03317=1236.829,159.897,-51.984,-177.725,5.664,148.314
C03318=1236.823,160.166,-52.008,-177.722,5.665,148.314
C03319=1236.819,160.436,-52.032,-177.720,5.666,148.313
C03320=1236.814,160.684,-52.054,-177.716,5.668,148.313
C03321=1236.809,160.933,-52.076,-177.714,5.669,148.312
C03322=1236.805,161.183,-52.097,-177.711,5.670,148.312
C03323=1236.800,161.432,-52.119,-177.709,5.671,148.311
C03324=1236.795,161.681,-52.141,-177.706,5.672,148.311
C03325=1236.791,161.930,-52.162,-177.704,5.674,148.310
C03326=1236.786,162.178,-52.184,-177.702,5.675,148.310
C03327=1236.781,162.428,-52.206,-177.699,5.676,148.309
C03328=1236.776,162.676,-52.228,-177.696,5.677,148.309
C03329=1236.772,162.926,-52.250,-177.693,5.679,148.308
C03330=1236.767,163.174,-52.272,-177.691,5.680,148.308
C03331=1236.763,163.424,-52.294,-177.689,5.681,148.308
C03332=1236.757,163.672,-52.316,-177.686,5.682,148.307
C03333=1236.753,163.922,-52.338,-177.684,5.683,148.307
C03334=1236.748,164.170,-52.360,-177.681,5.685,148.306
C03335=1236.744,164.420,-52.382,-177.679,5.686,148.306
C03336=1236.739,164.668,-52.403,-177.676,5.688,148.305
C03337=1236.734,164.917,-52.425,-177.673,5.688,148.305
C03338=1236.730,165.166,-52.447,-177.671,5.690,148.304
C03339=1236.725,165.415,-52.469,-177.668,5.691,148.304
C03340=1236.720,165.665,-52.491,-177.665,5.693,148.303
C03341=1236.715,165.913,-52.513,-177.663,5.694,148.303
C03342=1236.711,166.162,-52.536,-177.661,5.694,148.302
C03343=1236.707,166.411,-52.558,-177.658,5.696,148.302
C03344=1236.702,166.660,-52.580,-177.656,5.697,148.301
C03345=1236.697,166.909,-52.601,-177.653,5.699,148.301
C03346=1236.692,167.158,-52.624,-177.651,5.700,148.301
C03347=1236.688,167.408,-52.646,-177.648,5.701,148.300
C03348=1236.683,167.656,-52.668,-177.646,5.702,148.300
C03349=1236.679,167.906,-52.690,-177.643,5.704,148.299
C03350=1236.674,168.154,-52.712,-177.640,5.705,148.299
C03351=1236.669,168.403,-52.735,-177.638,5.706,148.298
C03352=1236.665,168.652,-52.756,-177.635,5.707,148.298
C03353=1236.660,168.901,-52.778,-177.632,5.709,148.297
C03354=1236.655,169.150,-52.800,-177.630,5.710,148.297
C03355=1236.651,169.399,-52.823,-177.627,5.712,148.296
C03356=1236.646,169.648,-52.845,-177.625,5.713,148.296
C03357=1236.642,169.897,-52.867,-177.622,5.714,148.296
C03358=1236.637,170.146,-52.889,-177.620,5.715,148.295
C03359=1236.632,170.395,-52.912,-177.617,5.717,148.295
C03360=1236.628,170.644,-52.934,-177.615,5.718,148.294
C03361=1236.623,170.893,-52.956,-177.612,5.719,148.294
C03362=1236.618,171.142,-52.979,-177.610,5.720,148.293
C03363=1236.613,171.390,-53.001,-177.607,5.722,148.293
C03364=1236.609,171.640,-53.023,-177.605,5.723,148.292
C03365=1236.604,171.889,-53.046,-177.602,5.725,148.292
C03366=1236.599,172.137,-53.068,-177.599,5.725,148.291
C03367=1236.595,172.387,-53.090,-177.597,5.727,148.291
C03368=1236.590,172.636,-53.112,-177.595,5.728,148.291
C03369=1236.586,172.884,-53.135,-177.592,5.730,148.290
C03370=1236.581,173.134,-53.157,-177.589,5.731,148.290
C03371=1236.576,173.383,-53.180,-177.587,5.733,148.289
C03372=1236.572,173.631,-53.202,-177.584,5.733,148.289
C03373=1236.567,173.880,-53.224,-177.582,5.735,148.288
C03374=1236.562,174.129,-53.247,-177.580,5.736,148.288
C03375=1236.558,174.378,-53.269,-177.576,5.738,148.287
C03376=1236.552,174.627,-53.292,-177.574,5.739,148.287
C03377=1236.548,174.876,-53.314,-177.572,5.741,148.287
C03378=1236.544,175.125,-53.336,-177.569,5.741,148.286
C03379=1236.539,175.374,-53.359,-177.566,5.743,148.286
C03380=1236.535,175.623,-53.382,-177.564,5.744,148.285
C03381=1236.530,175.872,-53.405,-177.561,5.746,148.285
C03382=1236.525,176.121,-53.427,-177.559,5.747,148.284
C03383=1236.520,176.370,-53.450,-177.556,5.749,148.284
C03384=1236.516,176.619,-53.472,-177.554,5.749,148.283
C03385=1236.511,176.867,-53.494,-177.551,5.751,148.283
C03386=1236.506,177.117,-53.517,-177.549,5.752,148.283
C03387=1236.502,177.365,-53.540,-177.546,5.754,148.282
C03388=1236.497,177.614,-53.562,-177.544,5.755,148.282
C03389=1236.493,177.863,-53.585,-177.541,5.756,148.281
C03390=1236.488,178.113,-53.607,-177.539,5.757,148.281
C03391=1236.483,178.361,-53.630,-177.536,5.759,148.280
C03392=1236.479,178.610,-53.653,-177.533,5.761,148.280
C03393=1236.474,178.859,-53.675,-177.531,5.762,148.280
C03394=1236.470,179.108,-53.699,-177.528,5.763,148.279
C03395=1236.465,179.357,-53.720,-177.526,5.764,148.279
C03396=1236.460,179.606,-53.744,-177.523,5.766,148.278
C03397=1236.456,179.855,-53.766,-177.521,5.767,148.278
C03398=1236.451,180.104,-53.789,-177.518,5.769,148.277
C03399=1236.447,180.352,-53.811,-177.516,5.770,148.277
C03400=1236.442,180.601,-53.835,-177.513,5.771,148.276
C03401=1236.437,180.851,-53.857,-177.511,5.772,148.276
C03402=1236.432,181.099,-53.880,-177.508,5.774,148.276
C03403=1236.428,181.348,-53.903,-177.505,5.776,148.275
C03404=1236.423,181.597,-53.925,-177.503,5.777,148.275
C03405=1236.419,181.846,-53.949,-177.500,5.779,148.274
C03406=1236.414,182.094,-53.971,-177.498,5.780,148.274
C03407=1236.409,182.343,-53.994,-177.495,5.781,148.273
C03408=1236.404,182.593,-54.017,-177.493,5.782,148.273
C03409=1236.400,182.842,-54.040,-177.490,5.784,148.273
C03410=1236.396,183.091,-54.063,-177.488,5.785,148.272
C03411=1236.390,183.339,-54.086,-177.485,5.787,148.272
C03412=1236.386,183.589,-54.108,-177.483,5.788,148.271
C03413=1236.381,183.838,-54.132,-177.480,5.789,148.271
C03414=1236.377,184.086,-54.154,-177.477,5.791,148.270
C03415=1236.373,184.335,-54.178,-177.475,5.792,148.270
C03416=1236.367,184.584,-54.201,-177.473,5.794,148.270
C03417=1236.363,184.833,-54.223,-177.469,5.795,148.269
C03418=1236.358,185.082,-54.246,-177.467,5.796,148.269
C03419=1236.354,185.331,-54.269,-177.465,5.798,148.268
C03420=1236.349,185.601,-54.294,-177.462,5.799,148.268
C03421=1236.344,185.870,-54.319,-177.460,5.801,148.267
C03422=1236.339,186.140,-54.344,-177.457,5.803,148.267
C03423=1236.334,186.409,-54.370,-177.454,5.804,148.266
C03424=1236.329,186.659,-54.392,-177.452,5.805,148.266
C03425=1236.325,186.908,-54.415,-177.449,5.807,148.266
C03426=1236.320,187.157,-54.438,-177.446,5.808,148.265
C03427=1236.316,187.405,-54.461,-177.444,5.810,148.265
C03428=1236.311,187.654,-54.484,-177.441,5.811,148.264
C03429=1236.306,187.903,-54.508,-177.439,5.812,148.264
C03430=1236.301,188.152,-54.531,-177.436,5.814,148.263
C03431=1236.297,188.400,-54.554,-177.433,5.816,148.263
C03432=1236.293,188.649,-54.577,-177.431,5.817,148.263
C03433=1236.288,188.899,-54.600,-177.429,5.819,148.262
C03434=1236.283,189.148,-54.624,-177.426,5.819,148.262
C03435=1236.278,189.397,-54.647,-177.423,5.821,148.261
C03436=1236.274,189.645,-54.670,-177.421,5.823,148.261
C03437=1236.269,189.894,-54.693,-177.419,5.824,148.261
C03438=1236.264,190.143,-54.716,-177.416,5.826,148.260
C03439=1236.260,190.392,-54.740,-177.413,5.827,148.260
C03440=1236.255,190.641,-54.763,-177.411,5.828,148.259
C03441=1236.251,190.889,-54.786,-177.408,5.830,148.259
C03442=1236.246,191.138,-54.809,-177.406,5.831,148.258
C03443=1236.242,191.387,-54.833,-177.403,5.833,148.258
C03444=1236.237,191.636,-54.857,-177.400,5.835,148.258
C03445=1236.233,191.885,-54.880,-177.398,5.836,148.257
C03446=1236.228,192.134,-54.903,-177.395,5.837,148.257
C03447=1236.223,192.382,-54.926,-177.393,5.838,148.256
C03448=1236.218,192.631,-54.950,-177.390,5.840,148.256
C03449=1236.214,192.880,-54.972,-177.388,5.842,148.256
C03450=1236.210,193.128,-54.996,-177.385,5.843,148.255
C03451=1236.205,193.378,-55.020,-177.383,5.845,148.255
C03452=1236.200,193.627,-55.043,-177.380,5.846,148.254
C03453=1236.195,193.876,-55.067,-177.378,5.847,148.254
C03454=1236.191,194.125,-55.090,-177.375,5.849,148.254
C03455=1236.186,194.373,-55.114,-177.372,5.851,148.253
C03456=1236.182,194.622,-55.137,-177.370,5.852,148.253
C03457=1236.177,194.871,-55.161,-177.367,5.854,148.252
C03458=1236.172,195.120,-55.184,-177.365,5.855,148.252
C03459=1236.168,195.369,-55.207,-177.362,5.856,148.252
C03460=1236.163,195.618,-55.231,-177.360,5.858,148.251
C03461=1236.158,195.867,-55.255,-177.357,5.859,148.251
C03462=1236.154,196.116,-55.278,-177.355,5.861,148.250
C03463=1236.149,196.364,-55.302,-177.352,5.863,148.250
C03464=1236.145,196.613,-55.326,-177.350,5.864,148.249
C03465=1236.140,196.862,-55.349,-177.347,5.865,148.249
C03466=1236.136,197.111,-55.373,-177.344,5.867,148.249
C03467=1236.131,197.360,-55.396,-177.342,5.868,148.248
C03468=1236.126,197.609,-55.420,-177.340,5.870,148.248
C03469=1236.122,197.857,-55.444,-177.336,5.872,148.248
C03470=1236.117,198.106,-55.467,-177.334,5.873,148.247
C03471=1236.112,198.355,-55.491,-177.332,5.875,148.247
C03472=1236.108,198.603,-55.515,-177.329,5.876,148.246
C03473=1236.103,198.853,-55.538,-177.327,5.878,148.246
C03474=1236.099,199.101,-55.562,-177.324,5.879,148.246
C03475=1236.094,199.350,-55.585,-177.321,5.881,148.245
C03476=1236.090,199.600,-55.609,-177.319,5.882,148.245
C03477=1236.086,199.848,-55.633,-177.317,5.884,148.244
C03478=1236.081,200.097,-55.657,-177.314,5.886,148.244
C03479=1236.077,200.346,-55.681,-177.312,5.887,148.244
C03480=1236.072,200.595,-55.704,-177.309,5.888,148.243
C03481=1236.068,200.843,-55.728,-177.306,5.890,148.243
C03482=1236.062,201.092,-55.752,-177.304,5.891,148.242
C03483=1236.058,201.341,-55.776,-177.301,5.893,148.242
C03484=1236.053,201.590,-55.799,-177.299,5.895,148.242
C03485=1236.049,201.838,-55.824,-177.296,5.896,148.241
C03486=1236.044,202.087,-55.847,-177.294,5.897,148.241
C03487=1236.040,202.336,-55.871,-177.291,5.899,148.241
C03488=1236.035,202.585,-55.895,-177.288,5.901,148.240
C03489=1236.031,202.834,-55.919,-177.286,5.902,148.240
C03490=1236.026,203.083,-55.943,-177.284,5.904,148.239
C03491=1236.021,203.332,-55.967,-177.280,5.906,148.239
C03492=1236.017,203.580,-55.991,-177.278,5.907,148.239
C03493=1236.012,203.829,-56.014,-177.276,5.908,148.238
C03494=1236.008,204.077,-56.038,-177.273,5.910,148.238
C03495=1236.003,204.327,-56.063,-177.271,5.911,148.238
C03496=1235.998,204.576,-56.087,-177.268,5.913,148.237
C03497=1235.994,204.824,-56.111,-177.265,5.915,148.237
C03498=1235.990,205.073,-56.135,-177.263,5.917,148.236
C03499=1235.985,205.322,-56.158,-177.261,5.918,148.236
C03500=1235.980,205.570,-56.183,-177.258,5.920,148.236
C03501=1235.975,205.819,-56.207,-177.255,5.921,148.235
C03502=1235.971,206.069,-56.231,-177.253,5.922,148.235
C03503=1235.967,206.317,-56.255,-177.251,5.924,148.235
C03504=1235.962,206.566,-56.279,-177.248,5.926,148.234
C03505=1235.957,206.815,-56.303,-177.245,5.928,148.234
C03506=1235.953,207.063,-56.327,-177.243,5.929,148.233
C03507=1235.948,207.313,-56.352,-177.240,5.931,148.233
C03508=1235.944,207.561,-56.376,-177.238,5.932,148.233
C03509=1235.939,207.809,-56.400,-177.235,5.933,148.232
C03510=1235.935,208.058,-56.423,-177.233,5.935,148.232
C03511=1235.930,208.307,-56.448,-177.230,5.937,148.231
C03512=1235.926,208.556,-56.473,-177.227,5.939,148.231
C03513=1235.921,208.805,-56.497,-177.225,5.940,148.231
C03514=1235.916,209.053,-56.521,-177.222,5.942,148.230
C03515=1235.912,209.302,-56.545,-177.220,5.944,148.230
C03516=1235.907,209.551,-56.569,-177.217,5.945,148.230
C03517=1235.903,209.800,-56.594,-177.215,5.946,148.229
C03518=1235.898,210.049,-56.618,-177.212,5.948,148.229
C03519=1235.893,210.297,-56.642,-177.209,5.950,148.228
C03520=1235.889,210.546,-56.667,-177.207,5.952,148.228
C03521=1235.885,210.795,-56.691,-177.205,5.953,148.228
C03522=1235.879,211.044,-56.715,-177.202,5.955,148.227
C03523=1235.875,211.293,-56.739,-177.199,5.956,148.227
C03524=1235.870,211.563,-56.766,-177.197,5.958,148.227
C03525=1235.865,211.834,-56.793,-177.194,5.960,148.226
C03526=1235.860,212.104,-56.820,-177.191,5.962,148.226
C03527=1235.856,212.374,-56.845,-177.188,5.964,148.225
C03528=1235.850,212.623,-56.870,-177.186,5.966,148.225
C03529=1235.847,212.872,-56.894,-177.183,5.966,148.225
C03530=1235.841,213.121,-56.919,-177.181,5.968,148.224
C03531=1235.837,213.369,-56.943,-177.178,5.970,148.224
C03532=1235.833,213.619,-56.968,-177.175,5.972,148.224
C03533=1235.828,213.867,-56.992,-177.173,5.973,148.223
C03534=1235.823,214.116,-57.017,-177.171,5.975,148.223
C03535=1235.819,214.365,-57.041,-177.168,5.977,148.223
C03536=1235.814,214.613,-57.066,-177.165,5.978,148.222
C03537=1235.810,214.862,-57.090,-177.163,5.980,148.222
C03538=1235.805,215.111,-57.115,-177.161,5.981,148.221
C03539=1235.801,215.359,-57.140,-177.158,5.983,148.221
C03540=1235.796,215.608,-57.164,-177.155,5.985,148.221
C03541=1235.792,215.857,-57.189,-177.152,5.987,148.220
C03542=1235.787,216.106,-57.213,-177.150,5.988,148.220
C03543=1235.783,216.354,-57.237,-177.148,5.990,148.220
C03544=1235.778,216.604,-57.262,-177.145,5.991,148.219
C03545=1235.774,216.852,-57.287,-177.142,5.993,148.219
C03546=1235.769,217.100,-57.312,-177.140,5.994,148.219
C03547=1235.765,217.349,-57.336,-177.138,5.996,148.218
C03548=1235.760,217.598,-57.361,-177.135,5.998,148.218
C03549=1235.755,217.847,-57.386,-177.132,6.000,148.218
C03550=1235.751,218.096,-57.410,-177.130,6.002,148.217
C03551=1235.746,218.344,-57.435,-177.127,6.003,148.217
C03552=1235.742,218.593,-57.460,-177.125,6.004,148.216
C03553=1235.737,218.842,-57.485,-177.122,6.006,148.216
C03554=1235.732,219.091,-57.509,-177.119,6.008,148.216
C03555=1235.729,219.339,-57.534,-177.117,6.010,148.215
C03556=1235.724,219.588,-57.559,-177.115,6.011,148.215
C03557=1235.720,219.837,-57.584,-177.112,6.013,148.215
C03558=1235.715,220.086,-57.608,-177.109,6.015,148.214
C03559=1235.710,220.334,-57.634,-177.107,6.017,148.214
C03560=1235.706,220.583,-57.658,-177.104,6.019,148.214
C03561=1235.701,220.832,-57.683,-177.102,6.020,148.213
C03562=1235.697,221.080,-57.708,-177.099,6.022,148.213
C03563=1235.692,221.329,-57.733,-177.097,6.023,148.213
C03564=1235.688,221.578,-57.758,-177.094,6.025,148.212
C03565=1235.683,221.826,-57.783,-177.092,6.027,148.212
C03566=1235.679,222.076,-57.807,-177.090,6.028,148.212
C03567=1235.674,222.324,-57.833,-177.087,6.030,148.211
C03568=1235.669,222.572,-57.857,-177.084,6.032,148.211
C03569=1235.665,222.822,-57.882,-177.082,6.034,148.211
C03570=1235.661,223.070,-57.907,-177.079,6.035,148.210
C03571=1235.656,223.319,-57.932,-177.077,6.036,148.210
C03572=1235.651,223.567,-57.958,-177.074,6.038,148.209
C03573=1235.647,223.817,-57.983,-177.071,6.040,148.209
C03574=1235.643,224.064,-58.008,-177.069,6.042,148.209
C03575=1235.638,224.314,-58.033,-177.066,6.044,148.208
C03576=1235.633,224.562,-58.057,-177.063,6.046,148.208
C03577=1235.629,224.811,-58.083,-177.061,6.047,148.208
C03578=1235.624,225.060,-58.107,-177.059,6.049,148.207
C03579=1235.620,225.308,-58.133,-177.056,6.051,148.207
C03580=1235.615,225.557,-58.158,-177.053,6.052,148.207
C03581=1235.611,225.806,-58.183,-177.051,6.054,148.206
C03582=1235.606,226.054,-58.209,-177.049,6.055,148.206
C03583=1235.602,226.303,-58.233,-177.046,6.057,148.206
C03584=1235.597,226.551,-58.258,-177.044,6.059,148.205
C03585=1235.593,226.801,-58.283,-177.041,6.061,148.205
C03586=1235.588,227.049,-58.309,-177.038,6.063,148.205
C03587=1235.583,227.298,-58.334,-177.036,6.065,148.205
C03588=1235.579,227.546,-58.359,-177.034,6.066,148.204
C03589=1235.574,227.795,-58.385,-177.031,6.068,148.204
C03590=1235.570,228.044,-58.409,-177.028,6.070,148.203
C03591=1235.566,228.292,-58.435,-177.026,6.071,148.203
C03592=1235.561,228.541,-58.461,-177.023,6.073,148.203
C03593=1235.556,228.790,-58.485,-177.021,6.075,148.203
C03594=1235.552,229.039,-58.511,-177.018,6.076,148.202
C03595=1235.547,229.287,-58.536,-177.016,6.078,148.202
C03596=1235.543,229.536,-58.561,-177.013,6.080,148.202
C03597=1235.539,229.785,-58.587,-177.011,6.082,148.201
C03598=1235.534,230.033,-58.613,-177.008,6.084,148.201
C03599=1235.529,230.283,-58.638,-177.005,6.086,148.201
C03600=1235.525,230.530,-58.662,-177.003,6.087,148.200
C03601=1235.521,230.779,-58.688,-177.001,6.089,148.200
C03602=1235.517,231.028,-58.714,-176.998,6.090,148.200
C03603=1235.511,231.277,-58.739,-176.996,6.093,148.199
C03604=1235.507,231.526,-58.764,-176.993,6.095,148.199
C03605=1235.502,231.774,-58.790,-176.991,6.096,148.199
C03606=1235.498,232.022,-58.815,-176.989,6.097,148.198
C03607=1235.494,232.271,-58.841,-176.986,6.099,148.198
C03608=1235.489,232.520,-58.866,-176.983,6.101,148.198
C03609=1235.485,232.769,-58.892,-176.981,6.103,148.198
C03610=1235.480,233.018,-58.917,-176.978,6.105,148.197
C03611=1235.476,233.266,-58.943,-176.976,6.107,148.197
C03612=1235.471,233.514,-58.969,-176.973,6.109,148.197
C03613=1235.467,233.763,-58.994,-176.971,6.110,148.196
C03614=1235.462,234.011,-59.020,-176.968,6.112,148.196
C03615=1235.458,234.261,-59.045,-176.966,6.114,148.196
C03616=1235.452,234.509,-59.071,-176.963,6.115,148.195
C03617=1235.448,234.758,-59.096,-176.960,6.117,148.195
C03618=1235.444,235.007,-59.122,-176.958,6.119,148.195
C03619=1235.440,235.256,-59.148,-176.955,6.121,148.194
C03620=1235.435,235.504,-59.173,-176.953,6.122,148.194
C03621=1235.430,235.753,-59.199,-176.951,6.124,148.194
C03622=1235.426,236.001,-59.225,-176.948,6.126,148.193
C03623=1235.421,236.249,-59.250,-176.946,6.128,148.193
C03624=1235.417,236.498,-59.276,-176.943,6.130,148.193
C03625=1235.413,236.747,-59.302,-176.941,6.132,148.193
C03626=1235.408,236.995,-59.327,-176.938,6.134,148.192
C03627=1235.403,237.244,-59.353,-176.935,6.136,148.192
C03628=1235.398,237.516,-59.381,-176.933,6.138,148.192
C03629=1235.394,237.787,-59.410,-176.930,6.139,148.191
C03630=1235.389,238.059,-59.438,-176.928,6.141,148.191
C03631=1235.384,238.330,-59.466,-176.925,6.143,148.191
C03632=1235.379,238.579,-59.491,-176.922,6.145,148.190
C03633=1235.375,238.827,-59.517,-176.920,6.147,148.190
C03634=1235.371,239.076,-59.544,-176.917,6.149,148.190
C03635=1235.366,239.324,-59.569,-176.914,6.151,148.189
C03636=1235.361,239.573,-59.595,-176.912,6.153,148.189
C03637=1235.357,239.822,-59.621,-176.910,6.154,148.189
C03638=1235.353,240.070,-59.647,-176.907,6.156,148.188
C03639=1235.348,240.319,-59.672,-176.905,6.157,148.188
C03640=1235.343,240.568,-59.698,-176.902,6.159,148.188
C03641=1235.339,240.816,-59.725,-176.900,6.162,148.188
C03642=1235.335,241.065,-59.751,-176.897,6.163,148.187
C03643=1235.330,241.313,-59.776,-176.895,6.165,148.187
C03644=1235.325,241.562,-59.802,-176.892,6.167,148.187
C03645=1235.321,241.811,-59.828,-176.889,6.169,148.187
C03646=1235.317,242.059,-59.855,-176.887,6.170,148.186
C03647=1235.313,242.308,-59.880,-176.885,6.172,148.186
C03648=1235.307,242.556,-59.906,-176.882,6.174,148.186
